//     PlcTask Inputs/GVL_iXlinker.EtherCAT_Master_EPPxxxx.Beckhoff_EPP2xxx.Beckhoff_EPP2xxxEK1122.A_0083_EPP2817_0008_0018.DIG_Diag_Inputs_Channel_2.Diag_Input[1] <-> DIG Diag Inputs Channel 2/Diag Input 2
//     PlcTask Inputs/GVL_iXlinker.EtherCAT_Master_EPPxxxx.Beckhoff_EPP2xxx.Beckhoff_EPP2xxxEK1122.A_0083_EPP2817_0008_0018.DIG_Diag_Inputs_Channel_2.Diag_Input[2] <-> DIG Diag Inputs Channel 2/Diag Input 3
//     PlcTask Inputs/GVL_iXlinker.EtherCAT_Master_EPPxxxx.Beckhoff_EPP2xxx.Beckhoff_EPP2xxxEK1122.A_0083_EPP2817_0008_0018.DIG_Diag_Inputs_Channel_2.Diag_Input[3] <-> DIG Diag Inputs Channel 2/Diag Input 4
//     PlcTask Inputs/GVL_iXlinker.EtherCAT_Master_EPPxxxx.Beckhoff_EPP2xxx.Beckhoff_EPP2xxxEK1122.A_0083_EPP2817_0008_0018.DIG_Diag_Inputs_Channel_2.Diag_Input[4] <-> DIG Diag Inputs Channel 2/Diag Input 5
//     PlcTask Inputs/GVL_iXlinker.EtherCAT_Master_EPPxxxx.Beckhoff_EPP2xxx.Beckhoff_EPP2xxxEK1122.A_0083_EPP2817_0008_0018.DIG_Diag_Inputs_Channel_2.Diag_Input[5] <-> DIG Diag Inputs Channel 2/Diag Input 6
//     PlcTask Inputs/GVL_iXlinker.EtherCAT_Master_EPPxxxx.Beckhoff_EPP2xxx.Beckhoff_EPP2xxxEK1122.A_0083_EPP2817_0008_0018.DIG_Diag_Inputs_Channel_2.Diag_Input[6] <-> DIG Diag Inputs Channel 2/Diag Input 7
//     PlcTask Inputs/GVL_iXlinker.EtherCAT_Master_EPPxxxx.Beckhoff_EPP2xxx.Beckhoff_EPP2xxxEK1122.A_0083_EPP2817_0008_0018.DIG_Diag_Inputs_Channel_2.Diag_Input[7] <-> DIG Diag Inputs Channel 2/Diag Input 8
//     PlcTask Inputs/GVL_iXlinker.EtherCAT_Master_EPPxxxx.Beckhoff_EPP2xxx.Beckhoff_EPP2xxxEK1122.A_0083_EPP2817_0008_0018.DIG_Diag_Inputs_Channel_3.Diag_Input[0] <-> DIG Diag Inputs Channel 3/Diag Input 1
//     PlcTask Inputs/GVL_iXlinker.EtherCAT_Master_EPPxxxx.Beckhoff_EPP2xxx.Beckhoff_EPP2xxxEK1122.A_0083_EPP2817_0008_0018.DIG_Diag_Inputs_Channel_3.Diag_Input[1] <-> DIG Diag Inputs Channel 3/Diag Input 2
//     PlcTask Inputs/GVL_iXlinker.EtherCAT_Master_EPPxxxx.Beckhoff_EPP2xxx.Beckhoff_EPP2xxxEK1122.A_0083_EPP2817_0008_0018.DIG_Diag_Inputs_Channel_3.Diag_Input[2] <-> DIG Diag Inputs Channel 3/Diag Input 3
//     PlcTask Inputs/GVL_iXlinker.EtherCAT_Master_EPPxxxx.Beckhoff_EPP2xxx.Beckhoff_EPP2xxxEK1122.A_0083_EPP2817_0008_0018.DIG_Diag_Inputs_Channel_3.Diag_Input[3] <-> DIG Diag Inputs Channel 3/Diag Input 4
//     PlcTask Inputs/GVL_iXlinker.EtherCAT_Master_EPPxxxx.Beckhoff_EPP2xxx.Beckhoff_EPP2xxxEK1122.A_0083_EPP2817_0008_0018.DIG_Diag_Inputs_Channel_3.Diag_Input[4] <-> DIG Diag Inputs Channel 3/Diag Input 5
//     PlcTask Inputs/GVL_iXlinker.EtherCAT_Master_EPPxxxx.Beckhoff_EPP2xxx.Beckhoff_EPP2xxxEK1122.A_0083_EPP2817_0008_0018.DIG_Diag_Inputs_Channel_3.Diag_Input[5] <-> DIG Diag Inputs Channel 3/Diag Input 6
//     PlcTask Inputs/GVL_iXlinker.EtherCAT_Master_EPPxxxx.Beckhoff_EPP2xxx.Beckhoff_EPP2xxxEK1122.A_0083_EPP2817_0008_0018.DIG_Diag_Inputs_Channel_3.Diag_Input[6] <-> DIG Diag Inputs Channel 3/Diag Input 7
//     PlcTask Inputs/GVL_iXlinker.EtherCAT_Master_EPPxxxx.Beckhoff_EPP2xxx.Beckhoff_EPP2xxxEK1122.A_0083_EPP2817_0008_0018.DIG_Diag_Inputs_Channel_3.Diag_Input[7] <-> DIG Diag Inputs Channel 3/Diag Input 8
//     PlcTask Inputs/GVL_iXlinker.EtherCAT_Master_EPPxxxx.Beckhoff_EPP2xxx.Beckhoff_EPP2xxxEK1122.A_0083_EPP2817_0008_0018.DIG_Inputs_Device.Safe_state_active <-> DIG Inputs Device/Safe state active
//     PlcTask Inputs/GVL_iXlinker.EtherCAT_Master_EPPxxxx.Beckhoff_EPP2xxx.Beckhoff_EPP2xxxEK1122.A_0083_EPP2817_0008_0018.DIG_Inputs_Device.Error_channel[0] <-> DIG Inputs Device/Error channel 1
//     PlcTask Inputs/GVL_iXlinker.EtherCAT_Master_EPPxxxx.Beckhoff_EPP2xxx.Beckhoff_EPP2xxxEK1122.A_0083_EPP2817_0008_0018.DIG_Inputs_Device.Error_channel[1] <-> DIG Inputs Device/Error channel 2
//     PlcTask Inputs/GVL_iXlinker.EtherCAT_Master_EPPxxxx.Beckhoff_EPP2xxx.Beckhoff_EPP2xxxEK1122.A_0083_EPP2817_0008_0018.DIG_Inputs_Device.Error_channel[2] <-> DIG Inputs Device/Error channel 3
//     PlcTask Inputs/GVL_iXlinker.EtherCAT_Master_EPPxxxx.Beckhoff_EPP2xxx.Beckhoff_EPP2xxxEK1122.A_0083_EPP2817_0008_0018.DIG_Inputs_Device.Us_Undervoltage <-> DIG Inputs Device/Us Undervoltage
//     PlcTask Inputs/GVL_iXlinker.EtherCAT_Master_EPPxxxx.Beckhoff_EPP2xxx.Beckhoff_EPP2xxxEK1122.A_0083_EPP2817_0008_0018.DIG_Inputs_Device.Up_Undervoltage <-> DIG Inputs Device/Up Undervoltage
//     PlcTask Inputs/GVL_iXlinker.EtherCAT_Master_EPPxxxx.Beckhoff_EPP2xxx.Beckhoff_EPP2xxxEK1122.A_0083_EPP2817_0008_0018.DIG_Inputs_Device.Sync_error <-> DIG Inputs Device/Sync error
//     PlcTask Inputs/GVL_iXlinker.EtherCAT_Master_EPPxxxx.Beckhoff_EPP2xxx.Beckhoff_EPP2xxxEK1122.A_0083_EPP2817_0008_0018.DIG_Inputs_Device.TxPDO_Toggle <-> DIG Inputs Device/TxPDO Toggle
//     PlcTask Outputs/GVL_iXlinker.EtherCAT_Master_EPPxxxx.Beckhoff_EPP2xxx.Beckhoff_EPP2xxxEK1122.A_0083_EPP2817_0008_0018.DIG_Output_Channel_1.Output[0] <-> DIG Output Channel 1/Output 1
//     PlcTask Outputs/GVL_iXlinker.EtherCAT_Master_EPPxxxx.Beckhoff_EPP2xxx.Beckhoff_EPP2xxxEK1122.A_0083_EPP2817_0008_0018.DIG_Output_Channel_1.Output[1] <-> DIG Output Channel 1/Output 2
//     PlcTask Outputs/GVL_iXlinker.EtherCAT_Master_EPPxxxx.Beckhoff_EPP2xxx.Beckhoff_EPP2xxxEK1122.A_0083_EPP2817_0008_0018.DIG_Output_Channel_1.Output[2] <-> DIG Output Channel 1/Output 3
//     PlcTask Outputs/GVL_iXlinker.EtherCAT_Master_EPPxxxx.Beckhoff_EPP2xxx.Beckhoff_EPP2xxxEK1122.A_0083_EPP2817_0008_0018.DIG_Output_Channel_1.Output[3] <-> DIG Output Channel 1/Output 4
//     PlcTask Outputs/GVL_iXlinker.EtherCAT_Master_EPPxxxx.Beckhoff_EPP2xxx.Beckhoff_EPP2xxxEK1122.A_0083_EPP2817_0008_0018.DIG_Output_Channel_1.Output[4] <-> DIG Output Channel 1/Output 5
//     PlcTask Outputs/GVL_iXlinker.EtherCAT_Master_EPPxxxx.Beckhoff_EPP2xxx.Beckhoff_EPP2xxxEK1122.A_0083_EPP2817_0008_0018.DIG_Output_Channel_1.Output[5] <-> DIG Output Channel 1/Output 6
//     PlcTask Outputs/GVL_iXlinker.EtherCAT_Master_EPPxxxx.Beckhoff_EPP2xxx.Beckhoff_EPP2xxxEK1122.A_0083_EPP2817_0008_0018.DIG_Output_Channel_1.Output[6] <-> DIG Output Channel 1/Output 7
//     PlcTask Outputs/GVL_iXlinker.EtherCAT_Master_EPPxxxx.Beckhoff_EPP2xxx.Beckhoff_EPP2xxxEK1122.A_0083_EPP2817_0008_0018.DIG_Output_Channel_1.Output[7] <-> DIG Output Channel 1/Output 8
//     PlcTask Outputs/GVL_iXlinker.EtherCAT_Master_EPPxxxx.Beckhoff_EPP2xxx.Beckhoff_EPP2xxxEK1122.A_0083_EPP2817_0008_0018.DIG_Output_Channel_2.Output[0] <-> DIG Output Channel 2/Output 1
//     PlcTask Outputs/GVL_iXlinker.EtherCAT_Master_EPPxxxx.Beckhoff_EPP2xxx.Beckhoff_EPP2xxxEK1122.A_0083_EPP2817_0008_0018.DIG_Output_Channel_2.Output[1] <-> DIG Output Channel 2/Output 2
//     PlcTask Outputs/GVL_iXlinker.EtherCAT_Master_EPPxxxx.Beckhoff_EPP2xxx.Beckhoff_EPP2xxxEK1122.A_0083_EPP2817_0008_0018.DIG_Output_Channel_2.Output[2] <-> DIG Output Channel 2/Output 3
//     PlcTask Outputs/GVL_iXlinker.EtherCAT_Master_EPPxxxx.Beckhoff_EPP2xxx.Beckhoff_EPP2xxxEK1122.A_0083_EPP2817_0008_0018.DIG_Output_Channel_2.Output[3] <-> DIG Output Channel 2/Output 4
//     PlcTask Outputs/GVL_iXlinker.EtherCAT_Master_EPPxxxx.Beckhoff_EPP2xxx.Beckhoff_EPP2xxxEK1122.A_0083_EPP2817_0008_0018.DIG_Output_Channel_2.Output[4] <-> DIG Output Channel 2/Output 5
//     PlcTask Outputs/GVL_iXlinker.EtherCAT_Master_EPPxxxx.Beckhoff_EPP2xxx.Beckhoff_EPP2xxxEK1122.A_0083_EPP2817_0008_0018.DIG_Output_Channel_2.Output[5] <-> DIG Output Channel 2/Output 6
//     PlcTask Outputs/GVL_iXlinker.EtherCAT_Master_EPPxxxx.Beckhoff_EPP2xxx.Beckhoff_EPP2xxxEK1122.A_0083_EPP2817_0008_0018.DIG_Output_Channel_2.Output[6] <-> DIG Output Channel 2/Output 7
//     PlcTask Outputs/GVL_iXlinker.EtherCAT_Master_EPPxxxx.Beckhoff_EPP2xxx.Beckhoff_EPP2xxxEK1122.A_0083_EPP2817_0008_0018.DIG_Output_Channel_2.Output[7] <-> DIG Output Channel 2/Output 8
//     PlcTask Outputs/GVL_iXlinker.EtherCAT_Master_EPPxxxx.Beckhoff_EPP2xxx.Beckhoff_EPP2xxxEK1122.A_0083_EPP2817_0008_0018.DIG_Output_Channel_3.Output[0] <-> DIG Output Channel 3/Output 1
//     PlcTask Outputs/GVL_iXlinker.EtherCAT_Master_EPPxxxx.Beckhoff_EPP2xxx.Beckhoff_EPP2xxxEK1122.A_0083_EPP2817_0008_0018.DIG_Output_Channel_3.Output[1] <-> DIG Output Channel 3/Output 2
//     PlcTask Outputs/GVL_iXlinker.EtherCAT_Master_EPPxxxx.Beckhoff_EPP2xxx.Beckhoff_EPP2xxxEK1122.A_0083_EPP2817_0008_0018.DIG_Output_Channel_3.Output[2] <-> DIG Output Channel 3/Output 3
//     PlcTask Outputs/GVL_iXlinker.EtherCAT_Master_EPPxxxx.Beckhoff_EPP2xxx.Beckhoff_EPP2xxxEK1122.A_0083_EPP2817_0008_0018.DIG_Output_Channel_3.Output[3] <-> DIG Output Channel 3/Output 4
//     PlcTask Outputs/GVL_iXlinker.EtherCAT_Master_EPPxxxx.Beckhoff_EPP2xxx.Beckhoff_EPP2xxxEK1122.A_0083_EPP2817_0008_0018.DIG_Output_Channel_3.Output[4] <-> DIG Output Channel 3/Output 5
//     PlcTask Outputs/GVL_iXlinker.EtherCAT_Master_EPPxxxx.Beckhoff_EPP2xxx.Beckhoff_EPP2xxxEK1122.A_0083_EPP2817_0008_0018.DIG_Output_Channel_3.Output[5] <-> DIG Output Channel 3/Output 6
//     PlcTask Outputs/GVL_iXlinker.EtherCAT_Master_EPPxxxx.Beckhoff_EPP2xxx.Beckhoff_EPP2xxxEK1122.A_0083_EPP2817_0008_0018.DIG_Output_Channel_3.Output[6] <-> DIG Output Channel 3/Output 7
//     PlcTask Outputs/GVL_iXlinker.EtherCAT_Master_EPPxxxx.Beckhoff_EPP2xxx.Beckhoff_EPP2xxxEK1122.A_0083_EPP2817_0008_0018.DIG_Output_Channel_3.Output[7] <-> DIG Output Channel 3/Output 8
//     PlcTask Outputs/GVL_iXlinker.EtherCAT_Master_EPPxxxx.Beckhoff_EPP2xxx.Beckhoff_EPP2xxxEK1122.A_0083_EPP2817_0008_0018.DIG_Outputs_Device.Set_safe_state <-> DIG Outputs Device/Set safe state
//     PlcTask Outputs/GVL_iXlinker.EtherCAT_Master_EPPxxxx.Beckhoff_EPP2xxx.Beckhoff_EPP2xxxEK1122.A_0083_EPP2817_0008_0018.DIG_Outputs_Device.Reset_outputs <-> DIG Outputs Device/Reset outputs
//     PlcTask Inputs/GVL_iXlinker.EtherCAT_Master_EPPxxxx.Beckhoff_EPP2xxx.Beckhoff_EPP2xxxEK1122.A_0083_EPP2817_0008_0018.WcState.WcState <-> WcState/WcState
//     PlcTask Inputs/GVL_iXlinker.EtherCAT_Master_EPPxxxx.Beckhoff_EPP2xxx.Beckhoff_EPP2xxxEK1122.A_0083_EPP2817_0008_0018.WcState.InputToggle <-> WcState/InputToggle
//     PlcTask Inputs/GVL_iXlinker.EtherCAT_Master_EPPxxxx.Beckhoff_EPP2xxx.Beckhoff_EPP2xxxEK1122.A_0083_EPP2817_0008_0018.InfoData.AdsAddr <-> InfoData/AdsAddr
//     PlcTask Inputs/GVL_iXlinker.EtherCAT_Master_EPPxxxx.Beckhoff_EPP2xxx.Beckhoff_EPP2xxxEK1122.A_0083_EPP2817_0008_0018.InfoData.State <-> InfoData/State
//   PLC/PLC Instance <-> EtherCAT Master EPPxxxx/Beckhoff EPP3xxx
//     PlcTask Inputs/GVL_iXlinker.EtherCAT_Master_EPPxxxx.Beckhoff_EPP3xxx.InfoData.State <-> InfoData/State
//   PLC/PLC Instance <-> EtherCAT Master EPPxxxx/Beckhoff EPP3xxx/Beckhoff EPP3xxxEK1122
//     PlcTask Inputs/GVL_iXlinker.EtherCAT_Master_EPPxxxx.Beckhoff_EPP3xxx.Beckhoff_EPP3xxxEK1122.InfoData.State <-> InfoData/State
//   PLC/PLC Instance <-> EtherCAT Master EPPxxxx/Beckhoff EPP3xxx/Beckhoff EPP3xxxEK1122/Beckhoff EPP3xxxsub EK1100
//     PlcTask Inputs/GVL_iXlinker.EtherCAT_Master_EPPxxxx.Beckhoff_EPP3xxx.Beckhoff_EPP3xxxEK1122.Beckhoff_EPP3xxxsub_EK1100.InfoData.State <-> InfoData/State
//   PLC/PLC Instance <-> EtherCAT Master EPPxxxx/Beckhoff EPP3xxx/Beckhoff EPP3xxxEK1122/A_0001(EPP3174-0002-0016)
//     PlcTask Inputs/GVL_iXlinker.EtherCAT_Master_EPPxxxx.Beckhoff_EPP3xxx.Beckhoff_EPP3xxxEK1122.A_0001_EPP3174_0002_0016.AI_Standard_Channel_1.Status/Underrange <-> AI Standard Channel 1/Status/Underrange
//     PlcTask Inputs/GVL_iXlinker.EtherCAT_Master_EPPxxxx.Beckhoff_EPP3xxx.Beckhoff_EPP3xxxEK1122.A_0001_EPP3174_0002_0016.AI_Standard_Channel_2.Status/Underrange <-> AI Standard Channel 2/Status/Underrange
//     PlcTask Inputs/GVL_iXlinker.EtherCAT_Master_EPPxxxx.Beckhoff_EPP3xxx.Beckhoff_EPP3xxxEK1122.A_0001_EPP3174_0002_0016.AI_Standard_Channel_3.Status/Underrange <-> AI Standard Channel 3/Status/Underrange
//     PlcTask Inputs/GVL_iXlinker.EtherCAT_Master_EPPxxxx.Beckhoff_EPP3xxx.Beckhoff_EPP3xxxEK1122.A_0001_EPP3174_0002_0016.AI_Standard_Channel_4.Status/Underrange <-> AI Standard Channel 4/Status/Underrange
//     PlcTask Inputs/GVL_iXlinker.EtherCAT_Master_EPPxxxx.Beckhoff_EPP3xxx.Beckhoff_EPP3xxxEK1122.A_0001_EPP3174_0002_0016.AI_Standard_Channel_1.Status/Overrange <-> AI Standard Channel 1/Status/Overrange
//     PlcTask Inputs/GVL_iXlinker.EtherCAT_Master_EPPxxxx.Beckhoff_EPP3xxx.Beckhoff_EPP3xxxEK1122.A_0001_EPP3174_0002_0016.AI_Standard_Channel_2.Status/Overrange <-> AI Standard Channel 2/Status/Overrange
//     PlcTask Inputs/GVL_iXlinker.EtherCAT_Master_EPPxxxx.Beckhoff_EPP3xxx.Beckhoff_EPP3xxxEK1122.A_0001_EPP3174_0002_0016.AI_Standard_Channel_3.Status/Overrange <-> AI Standard Channel 3/Status/Overrange
//     PlcTask Inputs/GVL_iXlinker.EtherCAT_Master_EPPxxxx.Beckhoff_EPP3xxx.Beckhoff_EPP3xxxEK1122.A_0001_EPP3174_0002_0016.AI_Standard_Channel_4.Status/Overrange <-> AI Standard Channel 4/Status/Overrange
//     PlcTask Inputs/GVL_iXlinker.EtherCAT_Master_EPPxxxx.Beckhoff_EPP3xxx.Beckhoff_EPP3xxxEK1122.A_0001_EPP3174_0002_0016.AI_Standard_Channel_1.Status/Limit_1 <-> AI Standard Channel 1/Status/Limit 1
//     PlcTask Inputs/GVL_iXlinker.EtherCAT_Master_EPPxxxx.Beckhoff_EPP3xxx.Beckhoff_EPP3xxxEK1122.A_0001_EPP3174_0002_0016.AI_Standard_Channel_1.Status/Limit_2 <-> AI Standard Channel 1/Status/Limit 2
//     PlcTask Inputs/GVL_iXlinker.EtherCAT_Master_EPPxxxx.Beckhoff_EPP3xxx.Beckhoff_EPP3xxxEK1122.A_0001_EPP3174_0002_0016.AI_Standard_Channel_2.Status/Limit_1 <-> AI Standard Channel 2/Status/Limit 1
//     PlcTask Inputs/GVL_iXlinker.EtherCAT_Master_EPPxxxx.Beckhoff_EPP3xxx.Beckhoff_EPP3xxxEK1122.A_0001_EPP3174_0002_0016.AI_Standard_Channel_2.Status/Limit_2 <-> AI Standard Channel 2/Status/Limit 2
//     PlcTask Inputs/GVL_iXlinker.EtherCAT_Master_EPPxxxx.Beckhoff_EPP3xxx.Beckhoff_EPP3xxxEK1122.A_0001_EPP3174_0002_0016.AI_Standard_Channel_3.Status/Limit_1 <-> AI Standard Channel 3/Status/Limit 1
//     PlcTask Inputs/GVL_iXlinker.EtherCAT_Master_EPPxxxx.Beckhoff_EPP3xxx.Beckhoff_EPP3xxxEK1122.A_0001_EPP3174_0002_0016.AI_Standard_Channel_3.Status/Limit_2 <-> AI Standard Channel 3/Status/Limit 2
//     PlcTask Inputs/GVL_iXlinker.EtherCAT_Master_EPPxxxx.Beckhoff_EPP3xxx.Beckhoff_EPP3xxxEK1122.A_0001_EPP3174_0002_0016.AI_Standard_Channel_4.Status/Limit_1 <-> AI Standard Channel 4/Status/Limit 1
//     PlcTask Inputs/GVL_iXlinker.EtherCAT_Master_EPPxxxx.Beckhoff_EPP3xxx.Beckhoff_EPP3xxxEK1122.A_0001_EPP3174_0002_0016.AI_Standard_Channel_4.Status/Limit_2 <-> AI Standard Channel 4/Status/Limit 2
//     PlcTask Inputs/GVL_iXlinker.EtherCAT_Master_EPPxxxx.Beckhoff_EPP3xxx.Beckhoff_EPP3xxxEK1122.A_0001_EPP3174_0002_0016.AI_Standard_Channel_1.Status/Error <-> AI Standard Channel 1/Status/Error
//     PlcTask Inputs/GVL_iXlinker.EtherCAT_Master_EPPxxxx.Beckhoff_EPP3xxx.Beckhoff_EPP3xxxEK1122.A_0001_EPP3174_0002_0016.AI_Standard_Channel_2.Status/Error <-> AI Standard Channel 2/Status/Error
//     PlcTask Inputs/GVL_iXlinker.EtherCAT_Master_EPPxxxx.Beckhoff_EPP3xxx.Beckhoff_EPP3xxxEK1122.A_0001_EPP3174_0002_0016.AI_Standard_Channel_3.Status/Error <-> AI Standard Channel 3/Status/Error
//     PlcTask Inputs/GVL_iXlinker.EtherCAT_Master_EPPxxxx.Beckhoff_EPP3xxx.Beckhoff_EPP3xxxEK1122.A_0001_EPP3174_0002_0016.AI_Standard_Channel_4.Status/Error <-> AI Standard Channel 4/Status/Error
//     PlcTask Inputs/GVL_iXlinker.EtherCAT_Master_EPPxxxx.Beckhoff_EPP3xxx.Beckhoff_EPP3xxxEK1122.A_0001_EPP3174_0002_0016.AI_Standard_Channel_1.Status/Sync_error <-> AI Standard Channel 1/Status/Sync error
//     PlcTask Inputs/GVL_iXlinker.EtherCAT_Master_EPPxxxx.Beckhoff_EPP3xxx.Beckhoff_EPP3xxxEK1122.A_0001_EPP3174_0002_0016.AI_Standard_Channel_2.Status/Sync_error <-> AI Standard Channel 2/Status/Sync error
//     PlcTask Inputs/GVL_iXlinker.EtherCAT_Master_EPPxxxx.Beckhoff_EPP3xxx.Beckhoff_EPP3xxxEK1122.A_0001_EPP3174_0002_0016.AI_Standard_Channel_3.Status/Sync_error <-> AI Standard Channel 3/Status/Sync error
//     PlcTask Inputs/GVL_iXlinker.EtherCAT_Master_EPPxxxx.Beckhoff_EPP3xxx.Beckhoff_EPP3xxxEK1122.A_0001_EPP3174_0002_0016.AI_Standard_Channel_4.Status/Sync_error <-> AI Standard Channel 4/Status/Sync error
//     PlcTask Inputs/GVL_iXlinker.EtherCAT_Master_EPPxxxx.Beckhoff_EPP3xxx.Beckhoff_EPP3xxxEK1122.A_0001_EPP3174_0002_0016.AI_Standard_Channel_1.Status/TxPDO_State <-> AI Standard Channel 1/Status/TxPDO State
//     PlcTask Inputs/GVL_iXlinker.EtherCAT_Master_EPPxxxx.Beckhoff_EPP3xxx.Beckhoff_EPP3xxxEK1122.A_0001_EPP3174_0002_0016.AI_Standard_Channel_2.Status/TxPDO_State <-> AI Standard Channel 2/Status/TxPDO State
//     PlcTask Inputs/GVL_iXlinker.EtherCAT_Master_EPPxxxx.Beckhoff_EPP3xxx.Beckhoff_EPP3xxxEK1122.A_0001_EPP3174_0002_0016.AI_Standard_Channel_3.Status/TxPDO_State <-> AI Standard Channel 3/Status/TxPDO State
//     PlcTask Inputs/GVL_iXlinker.EtherCAT_Master_EPPxxxx.Beckhoff_EPP3xxx.Beckhoff_EPP3xxxEK1122.A_0001_EPP3174_0002_0016.AI_Standard_Channel_4.Status/TxPDO_State <-> AI Standard Channel 4/Status/TxPDO State
//     PlcTask Inputs/GVL_iXlinker.EtherCAT_Master_EPPxxxx.Beckhoff_EPP3xxx.Beckhoff_EPP3xxxEK1122.A_0001_EPP3174_0002_0016.AI_Standard_Channel_1.Status/TxPDO_Toggle <-> AI Standard Channel 1/Status/TxPDO Toggle
//     PlcTask Inputs/GVL_iXlinker.EtherCAT_Master_EPPxxxx.Beckhoff_EPP3xxx.Beckhoff_EPP3xxxEK1122.A_0001_EPP3174_0002_0016.AI_Standard_Channel_2.Status/TxPDO_Toggle <-> AI Standard Channel 2/Status/TxPDO Toggle
//     PlcTask Inputs/GVL_iXlinker.EtherCAT_Master_EPPxxxx.Beckhoff_EPP3xxx.Beckhoff_EPP3xxxEK1122.A_0001_EPP3174_0002_0016.AI_Standard_Channel_3.Status/TxPDO_Toggle <-> AI Standard Channel 3/Status/TxPDO Toggle
//     PlcTask Inputs/GVL_iXlinker.EtherCAT_Master_EPPxxxx.Beckhoff_EPP3xxx.Beckhoff_EPP3xxxEK1122.A_0001_EPP3174_0002_0016.AI_Standard_Channel_4.Status/TxPDO_Toggle <-> AI Standard Channel 4/Status/TxPDO Toggle
//     PlcTask Inputs/GVL_iXlinker.EtherCAT_Master_EPPxxxx.Beckhoff_EPP3xxx.Beckhoff_EPP3xxxEK1122.A_0001_EPP3174_0002_0016.AI_Standard_Channel_1.Value <-> AI Standard Channel 1/Value
//     PlcTask Inputs/GVL_iXlinker.EtherCAT_Master_EPPxxxx.Beckhoff_EPP3xxx.Beckhoff_EPP3xxxEK1122.A_0001_EPP3174_0002_0016.AI_Standard_Channel_2.Value <-> AI Standard Channel 2/Value
//     PlcTask Inputs/GVL_iXlinker.EtherCAT_Master_EPPxxxx.Beckhoff_EPP3xxx.Beckhoff_EPP3xxxEK1122.A_0001_EPP3174_0002_0016.AI_Standard_Channel_3.Value <-> AI Standard Channel 3/Value
//     PlcTask Inputs/GVL_iXlinker.EtherCAT_Master_EPPxxxx.Beckhoff_EPP3xxx.Beckhoff_EPP3xxxEK1122.A_0001_EPP3174_0002_0016.AI_Standard_Channel_4.Value <-> AI Standard Channel 4/Value
//     PlcTask Inputs/GVL_iXlinker.EtherCAT_Master_EPPxxxx.Beckhoff_EPP3xxx.Beckhoff_EPP3xxxEK1122.A_0001_EPP3174_0002_0016.WcState.WcState <-> WcState/WcState
//     PlcTask Inputs/GVL_iXlinker.EtherCAT_Master_EPPxxxx.Beckhoff_EPP3xxx.Beckhoff_EPP3xxxEK1122.A_0001_EPP3174_0002_0016.WcState.InputToggle <-> WcState/InputToggle
//     PlcTask Inputs/GVL_iXlinker.EtherCAT_Master_EPPxxxx.Beckhoff_EPP3xxx.Beckhoff_EPP3xxxEK1122.A_0001_EPP3174_0002_0016.InfoData.AdsAddr <-> InfoData/AdsAddr
//     PlcTask Inputs/GVL_iXlinker.EtherCAT_Master_EPPxxxx.Beckhoff_EPP3xxx.Beckhoff_EPP3xxxEK1122.A_0001_EPP3174_0002_0016.InfoData.State <-> InfoData/State
//   PLC/PLC Instance <-> EtherCAT Master EPPxxxx/Beckhoff EPP3xxx/Beckhoff EPP3xxxEK1122/A_0002(EPP3174-0002-0017)
//     PlcTask Inputs/GVL_iXlinker.EtherCAT_Master_EPPxxxx.Beckhoff_EPP3xxx.Beckhoff_EPP3xxxEK1122.A_0002_EPP3174_0002_0017.AI_Standard_Channel_1.Status/Underrange <-> AI Standard Channel 1/Status/Underrange
//     PlcTask Inputs/GVL_iXlinker.EtherCAT_Master_EPPxxxx.Beckhoff_EPP3xxx.Beckhoff_EPP3xxxEK1122.A_0002_EPP3174_0002_0017.AI_Standard_Channel_2.Status/Underrange <-> AI Standard Channel 2/Status/Underrange
//     PlcTask Inputs/GVL_iXlinker.EtherCAT_Master_EPPxxxx.Beckhoff_EPP3xxx.Beckhoff_EPP3xxxEK1122.A_0002_EPP3174_0002_0017.AI_Standard_Channel_3.Status/Underrange <-> AI Standard Channel 3/Status/Underrange
//     PlcTask Inputs/GVL_iXlinker.EtherCAT_Master_EPPxxxx.Beckhoff_EPP3xxx.Beckhoff_EPP3xxxEK1122.A_0002_EPP3174_0002_0017.AI_Standard_Channel_4.Status/Underrange <-> AI Standard Channel 4/Status/Underrange
//     PlcTask Inputs/GVL_iXlinker.EtherCAT_Master_EPPxxxx.Beckhoff_EPP3xxx.Beckhoff_EPP3xxxEK1122.A_0002_EPP3174_0002_0017.AI_Standard_Channel_1.Status/Overrange <-> AI Standard Channel 1/Status/Overrange
//     PlcTask Inputs/GVL_iXlinker.EtherCAT_Master_EPPxxxx.Beckhoff_EPP3xxx.Beckhoff_EPP3xxxEK1122.A_0002_EPP3174_0002_0017.AI_Standard_Channel_2.Status/Overrange <-> AI Standard Channel 2/Status/Overrange
//     PlcTask Inputs/GVL_iXlinker.EtherCAT_Master_EPPxxxx.Beckhoff_EPP3xxx.Beckhoff_EPP3xxxEK1122.A_0002_EPP3174_0002_0017.AI_Standard_Channel_3.Status/Overrange <-> AI Standard Channel 3/Status/Overrange
//     PlcTask Inputs/GVL_iXlinker.EtherCAT_Master_EPPxxxx.Beckhoff_EPP3xxx.Beckhoff_EPP3xxxEK1122.A_0002_EPP3174_0002_0017.AI_Standard_Channel_4.Status/Overrange <-> AI Standard Channel 4/Status/Overrange
//     PlcTask Inputs/GVL_iXlinker.EtherCAT_Master_EPPxxxx.Beckhoff_EPP3xxx.Beckhoff_EPP3xxxEK1122.A_0002_EPP3174_0002_0017.AI_Standard_Channel_1.Status/Limit_1 <-> AI Standard Channel 1/Status/Limit 1
//     PlcTask Inputs/GVL_iXlinker.EtherCAT_Master_EPPxxxx.Beckhoff_EPP3xxx.Beckhoff_EPP3xxxEK1122.A_0002_EPP3174_0002_0017.AI_Standard_Channel_1.Status/Limit_2 <-> AI Standard Channel 1/Status/Limit 2
//     PlcTask Inputs/GVL_iXlinker.EtherCAT_Master_EPPxxxx.Beckhoff_EPP3xxx.Beckhoff_EPP3xxxEK1122.A_0002_EPP3174_0002_0017.AI_Standard_Channel_2.Status/Limit_1 <-> AI Standard Channel 2/Status/Limit 1
//     PlcTask Inputs/GVL_iXlinker.EtherCAT_Master_EPPxxxx.Beckhoff_EPP3xxx.Beckhoff_EPP3xxxEK1122.A_0002_EPP3174_0002_0017.AI_Standard_Channel_2.Status/Limit_2 <-> AI Standard Channel 2/Status/Limit 2
//     PlcTask Inputs/GVL_iXlinker.EtherCAT_Master_EPPxxxx.Beckhoff_EPP3xxx.Beckhoff_EPP3xxxEK1122.A_0002_EPP3174_0002_0017.AI_Standard_Channel_3.Status/Limit_1 <-> AI Standard Channel 3/Status/Limit 1
//     PlcTask Inputs/GVL_iXlinker.EtherCAT_Master_EPPxxxx.Beckhoff_EPP3xxx.Beckhoff_EPP3xxxEK1122.A_0002_EPP3174_0002_0017.AI_Standard_Channel_3.Status/Limit_2 <-> AI Standard Channel 3/Status/Limit 2
//     PlcTask Inputs/GVL_iXlinker.EtherCAT_Master_EPPxxxx.Beckhoff_EPP3xxx.Beckhoff_EPP3xxxEK1122.A_0002_EPP3174_0002_0017.AI_Standard_Channel_4.Status/Limit_1 <-> AI Standard Channel 4/Status/Limit 1
//     PlcTask Inputs/GVL_iXlinker.EtherCAT_Master_EPPxxxx.Beckhoff_EPP3xxx.Beckhoff_EPP3xxxEK1122.A_0002_EPP3174_0002_0017.AI_Standard_Channel_4.Status/Limit_2 <-> AI Standard Channel 4/Status/Limit 2
//     PlcTask Inputs/GVL_iXlinker.EtherCAT_Master_EPPxxxx.Beckhoff_EPP3xxx.Beckhoff_EPP3xxxEK1122.A_0002_EPP3174_0002_0017.AI_Standard_Channel_1.Status/Error <-> AI Standard Channel 1/Status/Error
//     PlcTask Inputs/GVL_iXlinker.EtherCAT_Master_EPPxxxx.Beckhoff_EPP3xxx.Beckhoff_EPP3xxxEK1122.A_0002_EPP3174_0002_0017.AI_Standard_Channel_2.Status/Error <-> AI Standard Channel 2/Status/Error
//     PlcTask Inputs/GVL_iXlinker.EtherCAT_Master_EPPxxxx.Beckhoff_EPP3xxx.Beckhoff_EPP3xxxEK1122.A_0002_EPP3174_0002_0017.AI_Standard_Channel_3.Status/Error <-> AI Standard Channel 3/Status/Error
//     PlcTask Inputs/GVL_iXlinker.EtherCAT_Master_EPPxxxx.Beckhoff_EPP3xxx.Beckhoff_EPP3xxxEK1122.A_0002_EPP3174_0002_0017.AI_Standard_Channel_4.Status/Error <-> AI Standard Channel 4/Status/Error
//     PlcTask Inputs/GVL_iXlinker.EtherCAT_Master_EPPxxxx.Beckhoff_EPP3xxx.Beckhoff_EPP3xxxEK1122.A_0002_EPP3174_0002_0017.AI_Standard_Channel_1.Status/Sync_error <-> AI Standard Channel 1/Status/Sync error
//     PlcTask Inputs/GVL_iXlinker.EtherCAT_Master_EPPxxxx.Beckhoff_EPP3xxx.Beckhoff_EPP3xxxEK1122.A_0002_EPP3174_0002_0017.AI_Standard_Channel_2.Status/Sync_error <-> AI Standard Channel 2/Status/Sync error
//     PlcTask Inputs/GVL_iXlinker.EtherCAT_Master_EPPxxxx.Beckhoff_EPP3xxx.Beckhoff_EPP3xxxEK1122.A_0002_EPP3174_0002_0017.AI_Standard_Channel_3.Status/Sync_error <-> AI Standard Channel 3/Status/Sync error
//     PlcTask Inputs/GVL_iXlinker.EtherCAT_Master_EPPxxxx.Beckhoff_EPP3xxx.Beckhoff_EPP3xxxEK1122.A_0002_EPP3174_0002_0017.AI_Standard_Channel_4.Status/Sync_error <-> AI Standard Channel 4/Status/Sync error
//     PlcTask Inputs/GVL_iXlinker.EtherCAT_Master_EPPxxxx.Beckhoff_EPP3xxx.Beckhoff_EPP3xxxEK1122.A_0002_EPP3174_0002_0017.AI_Standard_Channel_1.Status/TxPDO_State <-> AI Standard Channel 1/Status/TxPDO State
//     PlcTask Inputs/GVL_iXlinker.EtherCAT_Master_EPPxxxx.Beckhoff_EPP3xxx.Beckhoff_EPP3xxxEK1122.A_0002_EPP3174_0002_0017.AI_Standard_Channel_2.Status/TxPDO_State <-> AI Standard Channel 2/Status/TxPDO State
//     PlcTask Inputs/GVL_iXlinker.EtherCAT_Master_EPPxxxx.Beckhoff_EPP3xxx.Beckhoff_EPP3xxxEK1122.A_0002_EPP3174_0002_0017.AI_Standard_Channel_3.Status/TxPDO_State <-> AI Standard Channel 3/Status/TxPDO State
//     PlcTask Inputs/GVL_iXlinker.EtherCAT_Master_EPPxxxx.Beckhoff_EPP3xxx.Beckhoff_EPP3xxxEK1122.A_0002_EPP3174_0002_0017.AI_Standard_Channel_4.Status/TxPDO_State <-> AI Standard Channel 4/Status/TxPDO State
//     PlcTask Inputs/GVL_iXlinker.EtherCAT_Master_EPPxxxx.Beckhoff_EPP3xxx.Beckhoff_EPP3xxxEK1122.A_0002_EPP3174_0002_0017.AI_Standard_Channel_1.Status/TxPDO_Toggle <-> AI Standard Channel 1/Status/TxPDO Toggle
//     PlcTask Inputs/GVL_iXlinker.EtherCAT_Master_EPPxxxx.Beckhoff_EPP3xxx.Beckhoff_EPP3xxxEK1122.A_0002_EPP3174_0002_0017.AI_Standard_Channel_2.Status/TxPDO_Toggle <-> AI Standard Channel 2/Status/TxPDO Toggle
//     PlcTask Inputs/GVL_iXlinker.EtherCAT_Master_EPPxxxx.Beckhoff_EPP3xxx.Beckhoff_EPP3xxxEK1122.A_0002_EPP3174_0002_0017.AI_Standard_Channel_3.Status/TxPDO_Toggle <-> AI Standard Channel 3/Status/TxPDO Toggle
//     PlcTask Inputs/GVL_iXlinker.EtherCAT_Master_EPPxxxx.Beckhoff_EPP3xxx.Beckhoff_EPP3xxxEK1122.A_0002_EPP3174_0002_0017.AI_Standard_Channel_4.Status/TxPDO_Toggle <-> AI Standard Channel 4/Status/TxPDO Toggle
//     PlcTask Inputs/GVL_iXlinker.EtherCAT_Master_EPPxxxx.Beckhoff_EPP3xxx.Beckhoff_EPP3xxxEK1122.A_0002_EPP3174_0002_0017.AI_Standard_Channel_1.Value <-> AI Standard Channel 1/Value
//     PlcTask Inputs/GVL_iXlinker.EtherCAT_Master_EPPxxxx.Beckhoff_EPP3xxx.Beckhoff_EPP3xxxEK1122.A_0002_EPP3174_0002_0017.AI_Standard_Channel_2.Value <-> AI Standard Channel 2/Value
//     PlcTask Inputs/GVL_iXlinker.EtherCAT_Master_EPPxxxx.Beckhoff_EPP3xxx.Beckhoff_EPP3xxxEK1122.A_0002_EPP3174_0002_0017.AI_Standard_Channel_3.Value <-> AI Standard Channel 3/Value
//     PlcTask Inputs/GVL_iXlinker.EtherCAT_Master_EPPxxxx.Beckhoff_EPP3xxx.Beckhoff_EPP3xxxEK1122.A_0002_EPP3174_0002_0017.AI_Standard_Channel_4.Value <-> AI Standard Channel 4/Value
//     PlcTask Inputs/GVL_iXlinker.EtherCAT_Master_EPPxxxx.Beckhoff_EPP3xxx.Beckhoff_EPP3xxxEK1122.A_0002_EPP3174_0002_0017.WcState.WcState <-> WcState/WcState
//     PlcTask Inputs/GVL_iXlinker.EtherCAT_Master_EPPxxxx.Beckhoff_EPP3xxx.Beckhoff_EPP3xxxEK1122.A_0002_EPP3174_0002_0017.WcState.InputToggle <-> WcState/InputToggle
//     PlcTask Inputs/GVL_iXlinker.EtherCAT_Master_EPPxxxx.Beckhoff_EPP3xxx.Beckhoff_EPP3xxxEK1122.A_0002_EPP3174_0002_0017.InfoData.AdsAddr <-> InfoData/AdsAddr
//     PlcTask Inputs/GVL_iXlinker.EtherCAT_Master_EPPxxxx.Beckhoff_EPP3xxx.Beckhoff_EPP3xxxEK1122.A_0002_EPP3174_0002_0017.InfoData.State <-> InfoData/State
//   PLC/PLC Instance <-> EtherCAT Master EPPxxxx/Beckhoff EPP3xxx/Beckhoff EPP3xxxEK1122/A_0003(EPP3174-0002-0018)
//     PlcTask Inputs/GVL_iXlinker.EtherCAT_Master_EPPxxxx.Beckhoff_EPP3xxx.Beckhoff_EPP3xxxEK1122.A_0003_EPP3174_0002_0018.AI_Standard_Channel_1.Status/Underrange <-> AI Standard Channel 1/Status/Underrange
//     PlcTask Inputs/GVL_iXlinker.EtherCAT_Master_EPPxxxx.Beckhoff_EPP3xxx.Beckhoff_EPP3xxxEK1122.A_0003_EPP3174_0002_0018.AI_Standard_Channel_2.Status/Underrange <-> AI Standard Channel 2/Status/Underrange
//     PlcTask Inputs/GVL_iXlinker.EtherCAT_Master_EPPxxxx.Beckhoff_EPP3xxx.Beckhoff_EPP3xxxEK1122.A_0003_EPP3174_0002_0018.AI_Standard_Channel_3.Status/Underrange <-> AI Standard Channel 3/Status/Underrange
//     PlcTask Inputs/GVL_iXlinker.EtherCAT_Master_EPPxxxx.Beckhoff_EPP3xxx.Beckhoff_EPP3xxxEK1122.A_0003_EPP3174_0002_0018.AI_Standard_Channel_4.Status/Underrange <-> AI Standard Channel 4/Status/Underrange
//     PlcTask Inputs/GVL_iXlinker.EtherCAT_Master_EPPxxxx.Beckhoff_EPP3xxx.Beckhoff_EPP3xxxEK1122.A_0003_EPP3174_0002_0018.AI_Standard_Channel_1.Status/Overrange <-> AI Standard Channel 1/Status/Overrange
//     PlcTask Inputs/GVL_iXlinker.EtherCAT_Master_EPPxxxx.Beckhoff_EPP3xxx.Beckhoff_EPP3xxxEK1122.A_0003_EPP3174_0002_0018.AI_Standard_Channel_2.Status/Overrange <-> AI Standard Channel 2/Status/Overrange
//     PlcTask Inputs/GVL_iXlinker.EtherCAT_Master_EPPxxxx.Beckhoff_EPP3xxx.Beckhoff_EPP3xxxEK1122.A_0003_EPP3174_0002_0018.AI_Standard_Channel_3.Status/Overrange <-> AI Standard Channel 3/Status/Overrange
//     PlcTask Inputs/GVL_iXlinker.EtherCAT_Master_EPPxxxx.Beckhoff_EPP3xxx.Beckhoff_EPP3xxxEK1122.A_0003_EPP3174_0002_0018.AI_Standard_Channel_4.Status/Overrange <-> AI Standard Channel 4/Status/Overrange
//     PlcTask Inputs/GVL_iXlinker.EtherCAT_Master_EPPxxxx.Beckhoff_EPP3xxx.Beckhoff_EPP3xxxEK1122.A_0003_EPP3174_0002_0018.AI_Standard_Channel_1.Status/Limit_1 <-> AI Standard Channel 1/Status/Limit 1
//     PlcTask Inputs/GVL_iXlinker.EtherCAT_Master_EPPxxxx.Beckhoff_EPP3xxx.Beckhoff_EPP3xxxEK1122.A_0003_EPP3174_0002_0018.AI_Standard_Channel_1.Status/Limit_2 <-> AI Standard Channel 1/Status/Limit 2
//     PlcTask Inputs/GVL_iXlinker.EtherCAT_Master_EPPxxxx.Beckhoff_EPP3xxx.Beckhoff_EPP3xxxEK1122.A_0003_EPP3174_0002_0018.AI_Standard_Channel_2.Status/Limit_1 <-> AI Standard Channel 2/Status/Limit 1
//     PlcTask Inputs/GVL_iXlinker.EtherCAT_Master_EPPxxxx.Beckhoff_EPP3xxx.Beckhoff_EPP3xxxEK1122.A_0003_EPP3174_0002_0018.AI_Standard_Channel_2.Status/Limit_2 <-> AI Standard Channel 2/Status/Limit 2
//     PlcTask Inputs/GVL_iXlinker.EtherCAT_Master_EPPxxxx.Beckhoff_EPP3xxx.Beckhoff_EPP3xxxEK1122.A_0003_EPP3174_0002_0018.AI_Standard_Channel_3.Status/Limit_1 <-> AI Standard Channel 3/Status/Limit 1
//     PlcTask Inputs/GVL_iXlinker.EtherCAT_Master_EPPxxxx.Beckhoff_EPP3xxx.Beckhoff_EPP3xxxEK1122.A_0003_EPP3174_0002_0018.AI_Standard_Channel_3.Status/Limit_2 <-> AI Standard Channel 3/Status/Limit 2
//     PlcTask Inputs/GVL_iXlinker.EtherCAT_Master_EPPxxxx.Beckhoff_EPP3xxx.Beckhoff_EPP3xxxEK1122.A_0003_EPP3174_0002_0018.AI_Standard_Channel_4.Status/Limit_1 <-> AI Standard Channel 4/Status/Limit 1
//     PlcTask Inputs/GVL_iXlinker.EtherCAT_Master_EPPxxxx.Beckhoff_EPP3xxx.Beckhoff_EPP3xxxEK1122.A_0003_EPP3174_0002_0018.AI_Standard_Channel_4.Status/Limit_2 <-> AI Standard Channel 4/Status/Limit 2
//     PlcTask Inputs/GVL_iXlinker.EtherCAT_Master_EPPxxxx.Beckhoff_EPP3xxx.Beckhoff_EPP3xxxEK1122.A_0003_EPP3174_0002_0018.AI_Standard_Channel_1.Status/Error <-> AI Standard Channel 1/Status/Error
//     PlcTask Inputs/GVL_iXlinker.EtherCAT_Master_EPPxxxx.Beckhoff_EPP3xxx.Beckhoff_EPP3xxxEK1122.A_0003_EPP3174_0002_0018.AI_Standard_Channel_2.Status/Error <-> AI Standard Channel 2/Status/Error
//     PlcTask Inputs/GVL_iXlinker.EtherCAT_Master_EPPxxxx.Beckhoff_EPP3xxx.Beckhoff_EPP3xxxEK1122.A_0003_EPP3174_0002_0018.AI_Standard_Channel_3.Status/Error <-> AI Standard Channel 3/Status/Error
//     PlcTask Inputs/GVL_iXlinker.EtherCAT_Master_EPPxxxx.Beckhoff_EPP3xxx.Beckhoff_EPP3xxxEK1122.A_0003_EPP3174_0002_0018.AI_Standard_Channel_4.Status/Error <-> AI Standard Channel 4/Status/Error
//     PlcTask Inputs/GVL_iXlinker.EtherCAT_Master_EPPxxxx.Beckhoff_EPP3xxx.Beckhoff_EPP3xxxEK1122.A_0003_EPP3174_0002_0018.AI_Standard_Channel_1.Status/Sync_error <-> AI Standard Channel 1/Status/Sync error
//     PlcTask Inputs/GVL_iXlinker.EtherCAT_Master_EPPxxxx.Beckhoff_EPP3xxx.Beckhoff_EPP3xxxEK1122.A_0003_EPP3174_0002_0018.AI_Standard_Channel_2.Status/Sync_error <-> AI Standard Channel 2/Status/Sync error
//     PlcTask Inputs/GVL_iXlinker.EtherCAT_Master_EPPxxxx.Beckhoff_EPP3xxx.Beckhoff_EPP3xxxEK1122.A_0003_EPP3174_0002_0018.AI_Standard_Channel_3.Status/Sync_error <-> AI Standard Channel 3/Status/Sync error
//     PlcTask Inputs/GVL_iXlinker.EtherCAT_Master_EPPxxxx.Beckhoff_EPP3xxx.Beckhoff_EPP3xxxEK1122.A_0003_EPP3174_0002_0018.AI_Standard_Channel_4.Status/Sync_error <-> AI Standard Channel 4/Status/Sync error
//     PlcTask Inputs/GVL_iXlinker.EtherCAT_Master_EPPxxxx.Beckhoff_EPP3xxx.Beckhoff_EPP3xxxEK1122.A_0003_EPP3174_0002_0018.AI_Standard_Channel_1.Status/TxPDO_State <-> AI Standard Channel 1/Status/TxPDO State
//     PlcTask Inputs/GVL_iXlinker.EtherCAT_Master_EPPxxxx.Beckhoff_EPP3xxx.Beckhoff_EPP3xxxEK1122.A_0003_EPP3174_0002_0018.AI_Standard_Channel_2.Status/TxPDO_State <-> AI Standard Channel 2/Status/TxPDO State
//     PlcTask Inputs/GVL_iXlinker.EtherCAT_Master_EPPxxxx.Beckhoff_EPP3xxx.Beckhoff_EPP3xxxEK1122.A_0003_EPP3174_0002_0018.AI_Standard_Channel_3.Status/TxPDO_State <-> AI Standard Channel 3/Status/TxPDO State
//     PlcTask Inputs/GVL_iXlinker.EtherCAT_Master_EPPxxxx.Beckhoff_EPP3xxx.Beckhoff_EPP3xxxEK1122.A_0003_EPP3174_0002_0018.AI_Standard_Channel_4.Status/TxPDO_State <-> AI Standard Channel 4/Status/TxPDO State
//     PlcTask Inputs/GVL_iXlinker.EtherCAT_Master_EPPxxxx.Beckhoff_EPP3xxx.Beckhoff_EPP3xxxEK1122.A_0003_EPP3174_0002_0018.AI_Standard_Channel_1.Status/TxPDO_Toggle <-> AI Standard Channel 1/Status/TxPDO Toggle
//     PlcTask Inputs/GVL_iXlinker.EtherCAT_Master_EPPxxxx.Beckhoff_EPP3xxx.Beckhoff_EPP3xxxEK1122.A_0003_EPP3174_0002_0018.AI_Standard_Channel_2.Status/TxPDO_Toggle <-> AI Standard Channel 2/Status/TxPDO Toggle
//     PlcTask Inputs/GVL_iXlinker.EtherCAT_Master_EPPxxxx.Beckhoff_EPP3xxx.Beckhoff_EPP3xxxEK1122.A_0003_EPP3174_0002_0018.AI_Standard_Channel_3.Status/TxPDO_Toggle <-> AI Standard Channel 3/Status/TxPDO Toggle
//     PlcTask Inputs/GVL_iXlinker.EtherCAT_Master_EPPxxxx.Beckhoff_EPP3xxx.Beckhoff_EPP3xxxEK1122.A_0003_EPP3174_0002_0018.AI_Standard_Channel_4.Status/TxPDO_Toggle <-> AI Standard Channel 4/Status/TxPDO Toggle
//     PlcTask Inputs/GVL_iXlinker.EtherCAT_Master_EPPxxxx.Beckhoff_EPP3xxx.Beckhoff_EPP3xxxEK1122.A_0003_EPP3174_0002_0018.AI_Standard_Channel_1.Value <-> AI Standard Channel 1/Value
//     PlcTask Inputs/GVL_iXlinker.EtherCAT_Master_EPPxxxx.Beckhoff_EPP3xxx.Beckhoff_EPP3xxxEK1122.A_0003_EPP3174_0002_0018.AI_Standard_Channel_2.Value <-> AI Standard Channel 2/Value
//     PlcTask Inputs/GVL_iXlinker.EtherCAT_Master_EPPxxxx.Beckhoff_EPP3xxx.Beckhoff_EPP3xxxEK1122.A_0003_EPP3174_0002_0018.AI_Standard_Channel_3.Value <-> AI Standard Channel 3/Value
//     PlcTask Inputs/GVL_iXlinker.EtherCAT_Master_EPPxxxx.Beckhoff_EPP3xxx.Beckhoff_EPP3xxxEK1122.A_0003_EPP3174_0002_0018.AI_Standard_Channel_4.Value <-> AI Standard Channel 4/Value
//     PlcTask Inputs/GVL_iXlinker.EtherCAT_Master_EPPxxxx.Beckhoff_EPP3xxx.Beckhoff_EPP3xxxEK1122.A_0003_EPP3174_0002_0018.WcState.WcState <-> WcState/WcState
//     PlcTask Inputs/GVL_iXlinker.EtherCAT_Master_EPPxxxx.Beckhoff_EPP3xxx.Beckhoff_EPP3xxxEK1122.A_0003_EPP3174_0002_0018.WcState.InputToggle <-> WcState/InputToggle
//     PlcTask Inputs/GVL_iXlinker.EtherCAT_Master_EPPxxxx.Beckhoff_EPP3xxx.Beckhoff_EPP3xxxEK1122.A_0003_EPP3174_0002_0018.InfoData.AdsAddr <-> InfoData/AdsAddr
//     PlcTask Inputs/GVL_iXlinker.EtherCAT_Master_EPPxxxx.Beckhoff_EPP3xxx.Beckhoff_EPP3xxxEK1122.A_0003_EPP3174_0002_0018.InfoData.State <-> InfoData/State
//   PLC/PLC Instance <-> EtherCAT Master EPPxxxx/Beckhoff EPP3xxx/Beckhoff EPP3xxxEK1122/A_0004(EPP3184-0002-0016)
//     PlcTask Inputs/GVL_iXlinker.EtherCAT_Master_EPPxxxx.Beckhoff_EPP3xxx.Beckhoff_EPP3xxxEK1122.A_0004_EPP3184_0002_0016.AI_Standard_Channel_1.Status/Underrange <-> AI Standard Channel 1/Status/Underrange
//     PlcTask Inputs/GVL_iXlinker.EtherCAT_Master_EPPxxxx.Beckhoff_EPP3xxx.Beckhoff_EPP3xxxEK1122.A_0004_EPP3184_0002_0016.AI_Standard_Channel_2.Status/Underrange <-> AI Standard Channel 2/Status/Underrange
//     PlcTask Inputs/GVL_iXlinker.EtherCAT_Master_EPPxxxx.Beckhoff_EPP3xxx.Beckhoff_EPP3xxxEK1122.A_0004_EPP3184_0002_0016.AI_Standard_Channel_3.Status/Underrange <-> AI Standard Channel 3/Status/Underrange
//     PlcTask Inputs/GVL_iXlinker.EtherCAT_Master_EPPxxxx.Beckhoff_EPP3xxx.Beckhoff_EPP3xxxEK1122.A_0004_EPP3184_0002_0016.AI_Standard_Channel_4.Status/Underrange <-> AI Standard Channel 4/Status/Underrange
//     PlcTask Inputs/GVL_iXlinker.EtherCAT_Master_EPPxxxx.Beckhoff_EPP3xxx.Beckhoff_EPP3xxxEK1122.A_0004_EPP3184_0002_0016.AI_Standard_Channel_1.Status/Overrange <-> AI Standard Channel 1/Status/Overrange
//     PlcTask Inputs/GVL_iXlinker.EtherCAT_Master_EPPxxxx.Beckhoff_EPP3xxx.Beckhoff_EPP3xxxEK1122.A_0004_EPP3184_0002_0016.AI_Standard_Channel_2.Status/Overrange <-> AI Standard Channel 2/Status/Overrange
//     PlcTask Inputs/GVL_iXlinker.EtherCAT_Master_EPPxxxx.Beckhoff_EPP3xxx.Beckhoff_EPP3xxxEK1122.A_0004_EPP3184_0002_0016.AI_Standard_Channel_3.Status/Overrange <-> AI Standard Channel 3/Status/Overrange
//     PlcTask Inputs/GVL_iXlinker.EtherCAT_Master_EPPxxxx.Beckhoff_EPP3xxx.Beckhoff_EPP3xxxEK1122.A_0004_EPP3184_0002_0016.AI_Standard_Channel_4.Status/Overrange <-> AI Standard Channel 4/Status/Overrange
//     PlcTask Inputs/GVL_iXlinker.EtherCAT_Master_EPPxxxx.Beckhoff_EPP3xxx.Beckhoff_EPP3xxxEK1122.A_0004_EPP3184_0002_0016.AI_Standard_Channel_1.Status/Limit_1 <-> AI Standard Channel 1/Status/Limit 1
//     PlcTask Inputs/GVL_iXlinker.EtherCAT_Master_EPPxxxx.Beckhoff_EPP3xxx.Beckhoff_EPP3xxxEK1122.A_0004_EPP3184_0002_0016.AI_Standard_Channel_1.Status/Limit_2 <-> AI Standard Channel 1/Status/Limit 2
//     PlcTask Inputs/GVL_iXlinker.EtherCAT_Master_EPPxxxx.Beckhoff_EPP3xxx.Beckhoff_EPP3xxxEK1122.A_0004_EPP3184_0002_0016.AI_Standard_Channel_2.Status/Limit_1 <-> AI Standard Channel 2/Status/Limit 1
//     PlcTask Inputs/GVL_iXlinker.EtherCAT_Master_EPPxxxx.Beckhoff_EPP3xxx.Beckhoff_EPP3xxxEK1122.A_0004_EPP3184_0002_0016.AI_Standard_Channel_2.Status/Limit_2 <-> AI Standard Channel 2/Status/Limit 2
//     PlcTask Inputs/GVL_iXlinker.EtherCAT_Master_EPPxxxx.Beckhoff_EPP3xxx.Beckhoff_EPP3xxxEK1122.A_0004_EPP3184_0002_0016.AI_Standard_Channel_3.Status/Limit_1 <-> AI Standard Channel 3/Status/Limit 1
//     PlcTask Inputs/GVL_iXlinker.EtherCAT_Master_EPPxxxx.Beckhoff_EPP3xxx.Beckhoff_EPP3xxxEK1122.A_0004_EPP3184_0002_0016.AI_Standard_Channel_3.Status/Limit_2 <-> AI Standard Channel 3/Status/Limit 2
//     PlcTask Inputs/GVL_iXlinker.EtherCAT_Master_EPPxxxx.Beckhoff_EPP3xxx.Beckhoff_EPP3xxxEK1122.A_0004_EPP3184_0002_0016.AI_Standard_Channel_4.Status/Limit_1 <-> AI Standard Channel 4/Status/Limit 1
//     PlcTask Inputs/GVL_iXlinker.EtherCAT_Master_EPPxxxx.Beckhoff_EPP3xxx.Beckhoff_EPP3xxxEK1122.A_0004_EPP3184_0002_0016.AI_Standard_Channel_4.Status/Limit_2 <-> AI Standard Channel 4/Status/Limit 2
//     PlcTask Inputs/GVL_iXlinker.EtherCAT_Master_EPPxxxx.Beckhoff_EPP3xxx.Beckhoff_EPP3xxxEK1122.A_0004_EPP3184_0002_0016.AI_Standard_Channel_1.Status/Error <-> AI Standard Channel 1/Status/Error
//     PlcTask Inputs/GVL_iXlinker.EtherCAT_Master_EPPxxxx.Beckhoff_EPP3xxx.Beckhoff_EPP3xxxEK1122.A_0004_EPP3184_0002_0016.AI_Standard_Channel_2.Status/Error <-> AI Standard Channel 2/Status/Error
//     PlcTask Inputs/GVL_iXlinker.EtherCAT_Master_EPPxxxx.Beckhoff_EPP3xxx.Beckhoff_EPP3xxxEK1122.A_0004_EPP3184_0002_0016.AI_Standard_Channel_3.Status/Error <-> AI Standard Channel 3/Status/Error
//     PlcTask Inputs/GVL_iXlinker.EtherCAT_Master_EPPxxxx.Beckhoff_EPP3xxx.Beckhoff_EPP3xxxEK1122.A_0004_EPP3184_0002_0016.AI_Standard_Channel_4.Status/Error <-> AI Standard Channel 4/Status/Error
//     PlcTask Inputs/GVL_iXlinker.EtherCAT_Master_EPPxxxx.Beckhoff_EPP3xxx.Beckhoff_EPP3xxxEK1122.A_0004_EPP3184_0002_0016.AI_Standard_Channel_1.Status/Sync_error <-> AI Standard Channel 1/Status/Sync error
//     PlcTask Inputs/GVL_iXlinker.EtherCAT_Master_EPPxxxx.Beckhoff_EPP3xxx.Beckhoff_EPP3xxxEK1122.A_0004_EPP3184_0002_0016.AI_Standard_Channel_2.Status/Sync_error <-> AI Standard Channel 2/Status/Sync error
//     PlcTask Inputs/GVL_iXlinker.EtherCAT_Master_EPPxxxx.Beckhoff_EPP3xxx.Beckhoff_EPP3xxxEK1122.A_0004_EPP3184_0002_0016.AI_Standard_Channel_3.Status/Sync_error <-> AI Standard Channel 3/Status/Sync error
//     PlcTask Inputs/GVL_iXlinker.EtherCAT_Master_EPPxxxx.Beckhoff_EPP3xxx.Beckhoff_EPP3xxxEK1122.A_0004_EPP3184_0002_0016.AI_Standard_Channel_4.Status/Sync_error <-> AI Standard Channel 4/Status/Sync error
//     PlcTask Inputs/GVL_iXlinker.EtherCAT_Master_EPPxxxx.Beckhoff_EPP3xxx.Beckhoff_EPP3xxxEK1122.A_0004_EPP3184_0002_0016.AI_Standard_Channel_1.Status/TxPDO_State <-> AI Standard Channel 1/Status/TxPDO State
//     PlcTask Inputs/GVL_iXlinker.EtherCAT_Master_EPPxxxx.Beckhoff_EPP3xxx.Beckhoff_EPP3xxxEK1122.A_0004_EPP3184_0002_0016.AI_Standard_Channel_2.Status/TxPDO_State <-> AI Standard Channel 2/Status/TxPDO State
//     PlcTask Inputs/GVL_iXlinker.EtherCAT_Master_EPPxxxx.Beckhoff_EPP3xxx.Beckhoff_EPP3xxxEK1122.A_0004_EPP3184_0002_0016.AI_Standard_Channel_3.Status/TxPDO_State <-> AI Standard Channel 3/Status/TxPDO State
//     PlcTask Inputs/GVL_iXlinker.EtherCAT_Master_EPPxxxx.Beckhoff_EPP3xxx.Beckhoff_EPP3xxxEK1122.A_0004_EPP3184_0002_0016.AI_Standard_Channel_4.Status/TxPDO_State <-> AI Standard Channel 4/Status/TxPDO State
//     PlcTask Inputs/GVL_iXlinker.EtherCAT_Master_EPPxxxx.Beckhoff_EPP3xxx.Beckhoff_EPP3xxxEK1122.A_0004_EPP3184_0002_0016.AI_Standard_Channel_1.Status/TxPDO_Toggle <-> AI Standard Channel 1/Status/TxPDO Toggle
//     PlcTask Inputs/GVL_iXlinker.EtherCAT_Master_EPPxxxx.Beckhoff_EPP3xxx.Beckhoff_EPP3xxxEK1122.A_0004_EPP3184_0002_0016.AI_Standard_Channel_2.Status/TxPDO_Toggle <-> AI Standard Channel 2/Status/TxPDO Toggle
//     PlcTask Inputs/GVL_iXlinker.EtherCAT_Master_EPPxxxx.Beckhoff_EPP3xxx.Beckhoff_EPP3xxxEK1122.A_0004_EPP3184_0002_0016.AI_Standard_Channel_3.Status/TxPDO_Toggle <-> AI Standard Channel 3/Status/TxPDO Toggle
//     PlcTask Inputs/GVL_iXlinker.EtherCAT_Master_EPPxxxx.Beckhoff_EPP3xxx.Beckhoff_EPP3xxxEK1122.A_0004_EPP3184_0002_0016.AI_Standard_Channel_4.Status/TxPDO_Toggle <-> AI Standard Channel 4/Status/TxPDO Toggle
//     PlcTask Inputs/GVL_iXlinker.EtherCAT_Master_EPPxxxx.Beckhoff_EPP3xxx.Beckhoff_EPP3xxxEK1122.A_0004_EPP3184_0002_0016.AI_Standard_Channel_1.Value <-> AI Standard Channel 1/Value
//     PlcTask Inputs/GVL_iXlinker.EtherCAT_Master_EPPxxxx.Beckhoff_EPP3xxx.Beckhoff_EPP3xxxEK1122.A_0004_EPP3184_0002_0016.AI_Standard_Channel_2.Value <-> AI Standard Channel 2/Value
//     PlcTask Inputs/GVL_iXlinker.EtherCAT_Master_EPPxxxx.Beckhoff_EPP3xxx.Beckhoff_EPP3xxxEK1122.A_0004_EPP3184_0002_0016.AI_Standard_Channel_3.Value <-> AI Standard Channel 3/Value
//     PlcTask Inputs/GVL_iXlinker.EtherCAT_Master_EPPxxxx.Beckhoff_EPP3xxx.Beckhoff_EPP3xxxEK1122.A_0004_EPP3184_0002_0016.AI_Standard_Channel_4.Value <-> AI Standard Channel 4/Value
//     PlcTask Inputs/GVL_iXlinker.EtherCAT_Master_EPPxxxx.Beckhoff_EPP3xxx.Beckhoff_EPP3xxxEK1122.A_0004_EPP3184_0002_0016.WcState.WcState <-> WcState/WcState
//     PlcTask Inputs/GVL_iXlinker.EtherCAT_Master_EPPxxxx.Beckhoff_EPP3xxx.Beckhoff_EPP3xxxEK1122.A_0004_EPP3184_0002_0016.WcState.InputToggle <-> WcState/InputToggle
//     PlcTask Inputs/GVL_iXlinker.EtherCAT_Master_EPPxxxx.Beckhoff_EPP3xxx.Beckhoff_EPP3xxxEK1122.A_0004_EPP3184_0002_0016.InfoData.AdsAddr <-> InfoData/AdsAddr
//     PlcTask Inputs/GVL_iXlinker.EtherCAT_Master_EPPxxxx.Beckhoff_EPP3xxx.Beckhoff_EPP3xxxEK1122.A_0004_EPP3184_0002_0016.InfoData.State <-> InfoData/State
//   PLC/PLC Instance <-> EtherCAT Master EPPxxxx/Beckhoff EPP3xxx/Beckhoff EPP3xxxEK1122/A_0005(EPP3184-0002-0017)
//     PlcTask Inputs/GVL_iXlinker.EtherCAT_Master_EPPxxxx.Beckhoff_EPP3xxx.Beckhoff_EPP3xxxEK1122.A_0005_EPP3184_0002_0017.AI_Standard_Channel_1.Status/Underrange <-> AI Standard Channel 1/Status/Underrange
//     PlcTask Inputs/GVL_iXlinker.EtherCAT_Master_EPPxxxx.Beckhoff_EPP3xxx.Beckhoff_EPP3xxxEK1122.A_0005_EPP3184_0002_0017.AI_Standard_Channel_2.Status/Underrange <-> AI Standard Channel 2/Status/Underrange
//     PlcTask Inputs/GVL_iXlinker.EtherCAT_Master_EPPxxxx.Beckhoff_EPP3xxx.Beckhoff_EPP3xxxEK1122.A_0005_EPP3184_0002_0017.AI_Standard_Channel_3.Status/Underrange <-> AI Standard Channel 3/Status/Underrange
//     PlcTask Inputs/GVL_iXlinker.EtherCAT_Master_EPPxxxx.Beckhoff_EPP3xxx.Beckhoff_EPP3xxxEK1122.A_0005_EPP3184_0002_0017.AI_Standard_Channel_4.Status/Underrange <-> AI Standard Channel 4/Status/Underrange
//     PlcTask Inputs/GVL_iXlinker.EtherCAT_Master_EPPxxxx.Beckhoff_EPP3xxx.Beckhoff_EPP3xxxEK1122.A_0005_EPP3184_0002_0017.AI_Standard_Channel_1.Status/Overrange <-> AI Standard Channel 1/Status/Overrange
//     PlcTask Inputs/GVL_iXlinker.EtherCAT_Master_EPPxxxx.Beckhoff_EPP3xxx.Beckhoff_EPP3xxxEK1122.A_0005_EPP3184_0002_0017.AI_Standard_Channel_2.Status/Overrange <-> AI Standard Channel 2/Status/Overrange
//     PlcTask Inputs/GVL_iXlinker.EtherCAT_Master_EPPxxxx.Beckhoff_EPP3xxx.Beckhoff_EPP3xxxEK1122.A_0005_EPP3184_0002_0017.AI_Standard_Channel_3.Status/Overrange <-> AI Standard Channel 3/Status/Overrange
//     PlcTask Inputs/GVL_iXlinker.EtherCAT_Master_EPPxxxx.Beckhoff_EPP3xxx.Beckhoff_EPP3xxxEK1122.A_0005_EPP3184_0002_0017.AI_Standard_Channel_4.Status/Overrange <-> AI Standard Channel 4/Status/Overrange
//     PlcTask Inputs/GVL_iXlinker.EtherCAT_Master_EPPxxxx.Beckhoff_EPP3xxx.Beckhoff_EPP3xxxEK1122.A_0005_EPP3184_0002_0017.AI_Standard_Channel_1.Status/Limit_1 <-> AI Standard Channel 1/Status/Limit 1
//     PlcTask Inputs/GVL_iXlinker.EtherCAT_Master_EPPxxxx.Beckhoff_EPP3xxx.Beckhoff_EPP3xxxEK1122.A_0005_EPP3184_0002_0017.AI_Standard_Channel_1.Status/Limit_2 <-> AI Standard Channel 1/Status/Limit 2
//     PlcTask Inputs/GVL_iXlinker.EtherCAT_Master_EPPxxxx.Beckhoff_EPP3xxx.Beckhoff_EPP3xxxEK1122.A_0005_EPP3184_0002_0017.AI_Standard_Channel_2.Status/Limit_1 <-> AI Standard Channel 2/Status/Limit 1
//     PlcTask Inputs/GVL_iXlinker.EtherCAT_Master_EPPxxxx.Beckhoff_EPP3xxx.Beckhoff_EPP3xxxEK1122.A_0005_EPP3184_0002_0017.AI_Standard_Channel_2.Status/Limit_2 <-> AI Standard Channel 2/Status/Limit 2
//     PlcTask Inputs/GVL_iXlinker.EtherCAT_Master_EPPxxxx.Beckhoff_EPP3xxx.Beckhoff_EPP3xxxEK1122.A_0005_EPP3184_0002_0017.AI_Standard_Channel_3.Status/Limit_1 <-> AI Standard Channel 3/Status/Limit 1
//     PlcTask Inputs/GVL_iXlinker.EtherCAT_Master_EPPxxxx.Beckhoff_EPP3xxx.Beckhoff_EPP3xxxEK1122.A_0005_EPP3184_0002_0017.AI_Standard_Channel_3.Status/Limit_2 <-> AI Standard Channel 3/Status/Limit 2
//     PlcTask Inputs/GVL_iXlinker.EtherCAT_Master_EPPxxxx.Beckhoff_EPP3xxx.Beckhoff_EPP3xxxEK1122.A_0005_EPP3184_0002_0017.AI_Standard_Channel_4.Status/Limit_1 <-> AI Standard Channel 4/Status/Limit 1
//     PlcTask Inputs/GVL_iXlinker.EtherCAT_Master_EPPxxxx.Beckhoff_EPP3xxx.Beckhoff_EPP3xxxEK1122.A_0005_EPP3184_0002_0017.AI_Standard_Channel_4.Status/Limit_2 <-> AI Standard Channel 4/Status/Limit 2
//     PlcTask Inputs/GVL_iXlinker.EtherCAT_Master_EPPxxxx.Beckhoff_EPP3xxx.Beckhoff_EPP3xxxEK1122.A_0005_EPP3184_0002_0017.AI_Standard_Channel_1.Status/Error <-> AI Standard Channel 1/Status/Error
//     PlcTask Inputs/GVL_iXlinker.EtherCAT_Master_EPPxxxx.Beckhoff_EPP3xxx.Beckhoff_EPP3xxxEK1122.A_0005_EPP3184_0002_0017.AI_Standard_Channel_2.Status/Error <-> AI Standard Channel 2/Status/Error
//     PlcTask Inputs/GVL_iXlinker.EtherCAT_Master_EPPxxxx.Beckhoff_EPP3xxx.Beckhoff_EPP3xxxEK1122.A_0005_EPP3184_0002_0017.AI_Standard_Channel_3.Status/Error <-> AI Standard Channel 3/Status/Error
//     PlcTask Inputs/GVL_iXlinker.EtherCAT_Master_EPPxxxx.Beckhoff_EPP3xxx.Beckhoff_EPP3xxxEK1122.A_0005_EPP3184_0002_0017.AI_Standard_Channel_4.Status/Error <-> AI Standard Channel 4/Status/Error
//     PlcTask Inputs/GVL_iXlinker.EtherCAT_Master_EPPxxxx.Beckhoff_EPP3xxx.Beckhoff_EPP3xxxEK1122.A_0005_EPP3184_0002_0017.AI_Standard_Channel_1.Status/Sync_error <-> AI Standard Channel 1/Status/Sync error
//     PlcTask Inputs/GVL_iXlinker.EtherCAT_Master_EPPxxxx.Beckhoff_EPP3xxx.Beckhoff_EPP3xxxEK1122.A_0005_EPP3184_0002_0017.AI_Standard_Channel_2.Status/Sync_error <-> AI Standard Channel 2/Status/Sync error
//     PlcTask Inputs/GVL_iXlinker.EtherCAT_Master_EPPxxxx.Beckhoff_EPP3xxx.Beckhoff_EPP3xxxEK1122.A_0005_EPP3184_0002_0017.AI_Standard_Channel_3.Status/Sync_error <-> AI Standard Channel 3/Status/Sync error
//     PlcTask Inputs/GVL_iXlinker.EtherCAT_Master_EPPxxxx.Beckhoff_EPP3xxx.Beckhoff_EPP3xxxEK1122.A_0005_EPP3184_0002_0017.AI_Standard_Channel_4.Status/Sync_error <-> AI Standard Channel 4/Status/Sync error
//     PlcTask Inputs/GVL_iXlinker.EtherCAT_Master_EPPxxxx.Beckhoff_EPP3xxx.Beckhoff_EPP3xxxEK1122.A_0005_EPP3184_0002_0017.AI_Standard_Channel_1.Status/TxPDO_State <-> AI Standard Channel 1/Status/TxPDO State
//     PlcTask Inputs/GVL_iXlinker.EtherCAT_Master_EPPxxxx.Beckhoff_EPP3xxx.Beckhoff_EPP3xxxEK1122.A_0005_EPP3184_0002_0017.AI_Standard_Channel_2.Status/TxPDO_State <-> AI Standard Channel 2/Status/TxPDO State
//     PlcTask Inputs/GVL_iXlinker.EtherCAT_Master_EPPxxxx.Beckhoff_EPP3xxx.Beckhoff_EPP3xxxEK1122.A_0005_EPP3184_0002_0017.AI_Standard_Channel_3.Status/TxPDO_State <-> AI Standard Channel 3/Status/TxPDO State
//     PlcTask Inputs/GVL_iXlinker.EtherCAT_Master_EPPxxxx.Beckhoff_EPP3xxx.Beckhoff_EPP3xxxEK1122.A_0005_EPP3184_0002_0017.AI_Standard_Channel_4.Status/TxPDO_State <-> AI Standard Channel 4/Status/TxPDO State
//     PlcTask Inputs/GVL_iXlinker.EtherCAT_Master_EPPxxxx.Beckhoff_EPP3xxx.Beckhoff_EPP3xxxEK1122.A_0005_EPP3184_0002_0017.AI_Standard_Channel_1.Status/TxPDO_Toggle <-> AI Standard Channel 1/Status/TxPDO Toggle
//     PlcTask Inputs/GVL_iXlinker.EtherCAT_Master_EPPxxxx.Beckhoff_EPP3xxx.Beckhoff_EPP3xxxEK1122.A_0005_EPP3184_0002_0017.AI_Standard_Channel_2.Status/TxPDO_Toggle <-> AI Standard Channel 2/Status/TxPDO Toggle
//     PlcTask Inputs/GVL_iXlinker.EtherCAT_Master_EPPxxxx.Beckhoff_EPP3xxx.Beckhoff_EPP3xxxEK1122.A_0005_EPP3184_0002_0017.AI_Standard_Channel_3.Status/TxPDO_Toggle <-> AI Standard Channel 3/Status/TxPDO Toggle
//     PlcTask Inputs/GVL_iXlinker.EtherCAT_Master_EPPxxxx.Beckhoff_EPP3xxx.Beckhoff_EPP3xxxEK1122.A_0005_EPP3184_0002_0017.AI_Standard_Channel_4.Status/TxPDO_Toggle <-> AI Standard Channel 4/Status/TxPDO Toggle
//     PlcTask Inputs/GVL_iXlinker.EtherCAT_Master_EPPxxxx.Beckhoff_EPP3xxx.Beckhoff_EPP3xxxEK1122.A_0005_EPP3184_0002_0017.AI_Standard_Channel_1.Value <-> AI Standard Channel 1/Value
//     PlcTask Inputs/GVL_iXlinker.EtherCAT_Master_EPPxxxx.Beckhoff_EPP3xxx.Beckhoff_EPP3xxxEK1122.A_0005_EPP3184_0002_0017.AI_Standard_Channel_2.Value <-> AI Standard Channel 2/Value
//     PlcTask Inputs/GVL_iXlinker.EtherCAT_Master_EPPxxxx.Beckhoff_EPP3xxx.Beckhoff_EPP3xxxEK1122.A_0005_EPP3184_0002_0017.AI_Standard_Channel_3.Value <-> AI Standard Channel 3/Value
//     PlcTask Inputs/GVL_iXlinker.EtherCAT_Master_EPPxxxx.Beckhoff_EPP3xxx.Beckhoff_EPP3xxxEK1122.A_0005_EPP3184_0002_0017.AI_Standard_Channel_4.Value <-> AI Standard Channel 4/Value
//     PlcTask Inputs/GVL_iXlinker.EtherCAT_Master_EPPxxxx.Beckhoff_EPP3xxx.Beckhoff_EPP3xxxEK1122.A_0005_EPP3184_0002_0017.WcState.WcState <-> WcState/WcState
//     PlcTask Inputs/GVL_iXlinker.EtherCAT_Master_EPPxxxx.Beckhoff_EPP3xxx.Beckhoff_EPP3xxxEK1122.A_0005_EPP3184_0002_0017.WcState.InputToggle <-> WcState/InputToggle
//     PlcTask Inputs/GVL_iXlinker.EtherCAT_Master_EPPxxxx.Beckhoff_EPP3xxx.Beckhoff_EPP3xxxEK1122.A_0005_EPP3184_0002_0017.InfoData.AdsAddr <-> InfoData/AdsAddr
//     PlcTask Inputs/GVL_iXlinker.EtherCAT_Master_EPPxxxx.Beckhoff_EPP3xxx.Beckhoff_EPP3xxxEK1122.A_0005_EPP3184_0002_0017.InfoData.State <-> InfoData/State
//   PLC/PLC Instance <-> EtherCAT Master EPPxxxx/Beckhoff EPP3xxx/Beckhoff EPP3xxxEK1122/A_0006(EPP3184-0002-0018)
//     PlcTask Inputs/GVL_iXlinker.EtherCAT_Master_EPPxxxx.Beckhoff_EPP3xxx.Beckhoff_EPP3xxxEK1122.A_0006_EPP3184_0002_0018.AI_Standard_Channel_1.Status/Underrange <-> AI Standard Channel 1/Status/Underrange
//     PlcTask Inputs/GVL_iXlinker.EtherCAT_Master_EPPxxxx.Beckhoff_EPP3xxx.Beckhoff_EPP3xxxEK1122.A_0006_EPP3184_0002_0018.AI_Standard_Channel_2.Status/Underrange <-> AI Standard Channel 2/Status/Underrange
//     PlcTask Inputs/GVL_iXlinker.EtherCAT_Master_EPPxxxx.Beckhoff_EPP3xxx.Beckhoff_EPP3xxxEK1122.A_0006_EPP3184_0002_0018.AI_Standard_Channel_3.Status/Underrange <-> AI Standard Channel 3/Status/Underrange
//     PlcTask Inputs/GVL_iXlinker.EtherCAT_Master_EPPxxxx.Beckhoff_EPP3xxx.Beckhoff_EPP3xxxEK1122.A_0006_EPP3184_0002_0018.AI_Standard_Channel_4.Status/Underrange <-> AI Standard Channel 4/Status/Underrange
//     PlcTask Inputs/GVL_iXlinker.EtherCAT_Master_EPPxxxx.Beckhoff_EPP3xxx.Beckhoff_EPP3xxxEK1122.A_0006_EPP3184_0002_0018.AI_Standard_Channel_1.Status/Overrange <-> AI Standard Channel 1/Status/Overrange
//     PlcTask Inputs/GVL_iXlinker.EtherCAT_Master_EPPxxxx.Beckhoff_EPP3xxx.Beckhoff_EPP3xxxEK1122.A_0006_EPP3184_0002_0018.AI_Standard_Channel_2.Status/Overrange <-> AI Standard Channel 2/Status/Overrange
//     PlcTask Inputs/GVL_iXlinker.EtherCAT_Master_EPPxxxx.Beckhoff_EPP3xxx.Beckhoff_EPP3xxxEK1122.A_0006_EPP3184_0002_0018.AI_Standard_Channel_3.Status/Overrange <-> AI Standard Channel 3/Status/Overrange
//     PlcTask Inputs/GVL_iXlinker.EtherCAT_Master_EPPxxxx.Beckhoff_EPP3xxx.Beckhoff_EPP3xxxEK1122.A_0006_EPP3184_0002_0018.AI_Standard_Channel_4.Status/Overrange <-> AI Standard Channel 4/Status/Overrange
//     PlcTask Inputs/GVL_iXlinker.EtherCAT_Master_EPPxxxx.Beckhoff_EPP3xxx.Beckhoff_EPP3xxxEK1122.A_0006_EPP3184_0002_0018.AI_Standard_Channel_1.Status/Limit_1 <-> AI Standard Channel 1/Status/Limit 1
//     PlcTask Inputs/GVL_iXlinker.EtherCAT_Master_EPPxxxx.Beckhoff_EPP3xxx.Beckhoff_EPP3xxxEK1122.A_0006_EPP3184_0002_0018.AI_Standard_Channel_1.Status/Limit_2 <-> AI Standard Channel 1/Status/Limit 2
//     PlcTask Inputs/GVL_iXlinker.EtherCAT_Master_EPPxxxx.Beckhoff_EPP3xxx.Beckhoff_EPP3xxxEK1122.A_0006_EPP3184_0002_0018.AI_Standard_Channel_2.Status/Limit_1 <-> AI Standard Channel 2/Status/Limit 1
//     PlcTask Inputs/GVL_iXlinker.EtherCAT_Master_EPPxxxx.Beckhoff_EPP3xxx.Beckhoff_EPP3xxxEK1122.A_0006_EPP3184_0002_0018.AI_Standard_Channel_2.Status/Limit_2 <-> AI Standard Channel 2/Status/Limit 2
//     PlcTask Inputs/GVL_iXlinker.EtherCAT_Master_EPPxxxx.Beckhoff_EPP3xxx.Beckhoff_EPP3xxxEK1122.A_0006_EPP3184_0002_0018.AI_Standard_Channel_3.Status/Limit_1 <-> AI Standard Channel 3/Status/Limit 1
//     PlcTask Inputs/GVL_iXlinker.EtherCAT_Master_EPPxxxx.Beckhoff_EPP3xxx.Beckhoff_EPP3xxxEK1122.A_0006_EPP3184_0002_0018.AI_Standard_Channel_3.Status/Limit_2 <-> AI Standard Channel 3/Status/Limit 2
//     PlcTask Inputs/GVL_iXlinker.EtherCAT_Master_EPPxxxx.Beckhoff_EPP3xxx.Beckhoff_EPP3xxxEK1122.A_0006_EPP3184_0002_0018.AI_Standard_Channel_4.Status/Limit_1 <-> AI Standard Channel 4/Status/Limit 1
//     PlcTask Inputs/GVL_iXlinker.EtherCAT_Master_EPPxxxx.Beckhoff_EPP3xxx.Beckhoff_EPP3xxxEK1122.A_0006_EPP3184_0002_0018.AI_Standard_Channel_4.Status/Limit_2 <-> AI Standard Channel 4/Status/Limit 2
//     PlcTask Inputs/GVL_iXlinker.EtherCAT_Master_EPPxxxx.Beckhoff_EPP3xxx.Beckhoff_EPP3xxxEK1122.A_0006_EPP3184_0002_0018.AI_Standard_Channel_1.Status/Error <-> AI Standard Channel 1/Status/Error
//     PlcTask Inputs/GVL_iXlinker.EtherCAT_Master_EPPxxxx.Beckhoff_EPP3xxx.Beckhoff_EPP3xxxEK1122.A_0006_EPP3184_0002_0018.AI_Standard_Channel_2.Status/Error <-> AI Standard Channel 2/Status/Error
//     PlcTask Inputs/GVL_iXlinker.EtherCAT_Master_EPPxxxx.Beckhoff_EPP3xxx.Beckhoff_EPP3xxxEK1122.A_0006_EPP3184_0002_0018.AI_Standard_Channel_3.Status/Error <-> AI Standard Channel 3/Status/Error
//     PlcTask Inputs/GVL_iXlinker.EtherCAT_Master_EPPxxxx.Beckhoff_EPP3xxx.Beckhoff_EPP3xxxEK1122.A_0006_EPP3184_0002_0018.AI_Standard_Channel_4.Status/Error <-> AI Standard Channel 4/Status/Error
//     PlcTask Inputs/GVL_iXlinker.EtherCAT_Master_EPPxxxx.Beckhoff_EPP3xxx.Beckhoff_EPP3xxxEK1122.A_0006_EPP3184_0002_0018.AI_Standard_Channel_1.Status/Sync_error <-> AI Standard Channel 1/Status/Sync error
//     PlcTask Inputs/GVL_iXlinker.EtherCAT_Master_EPPxxxx.Beckhoff_EPP3xxx.Beckhoff_EPP3xxxEK1122.A_0006_EPP3184_0002_0018.AI_Standard_Channel_2.Status/Sync_error <-> AI Standard Channel 2/Status/Sync error
//     PlcTask Inputs/GVL_iXlinker.EtherCAT_Master_EPPxxxx.Beckhoff_EPP3xxx.Beckhoff_EPP3xxxEK1122.A_0006_EPP3184_0002_0018.AI_Standard_Channel_3.Status/Sync_error <-> AI Standard Channel 3/Status/Sync error
//     PlcTask Inputs/GVL_iXlinker.EtherCAT_Master_EPPxxxx.Beckhoff_EPP3xxx.Beckhoff_EPP3xxxEK1122.A_0006_EPP3184_0002_0018.AI_Standard_Channel_4.Status/Sync_error <-> AI Standard Channel 4/Status/Sync error
//     PlcTask Inputs/GVL_iXlinker.EtherCAT_Master_EPPxxxx.Beckhoff_EPP3xxx.Beckhoff_EPP3xxxEK1122.A_0006_EPP3184_0002_0018.AI_Standard_Channel_1.Status/TxPDO_State <-> AI Standard Channel 1/Status/TxPDO State
//     PlcTask Inputs/GVL_iXlinker.EtherCAT_Master_EPPxxxx.Beckhoff_EPP3xxx.Beckhoff_EPP3xxxEK1122.A_0006_EPP3184_0002_0018.AI_Standard_Channel_2.Status/TxPDO_State <-> AI Standard Channel 2/Status/TxPDO State
//     PlcTask Inputs/GVL_iXlinker.EtherCAT_Master_EPPxxxx.Beckhoff_EPP3xxx.Beckhoff_EPP3xxxEK1122.A_0006_EPP3184_0002_0018.AI_Standard_Channel_3.Status/TxPDO_State <-> AI Standard Channel 3/Status/TxPDO State
//     PlcTask Inputs/GVL_iXlinker.EtherCAT_Master_EPPxxxx.Beckhoff_EPP3xxx.Beckhoff_EPP3xxxEK1122.A_0006_EPP3184_0002_0018.AI_Standard_Channel_4.Status/TxPDO_State <-> AI Standard Channel 4/Status/TxPDO State
//     PlcTask Inputs/GVL_iXlinker.EtherCAT_Master_EPPxxxx.Beckhoff_EPP3xxx.Beckhoff_EPP3xxxEK1122.A_0006_EPP3184_0002_0018.AI_Standard_Channel_1.Status/TxPDO_Toggle <-> AI Standard Channel 1/Status/TxPDO Toggle
//     PlcTask Inputs/GVL_iXlinker.EtherCAT_Master_EPPxxxx.Beckhoff_EPP3xxx.Beckhoff_EPP3xxxEK1122.A_0006_EPP3184_0002_0018.AI_Standard_Channel_2.Status/TxPDO_Toggle <-> AI Standard Channel 2/Status/TxPDO Toggle
//     PlcTask Inputs/GVL_iXlinker.EtherCAT_Master_EPPxxxx.Beckhoff_EPP3xxx.Beckhoff_EPP3xxxEK1122.A_0006_EPP3184_0002_0018.AI_Standard_Channel_3.Status/TxPDO_Toggle <-> AI Standard Channel 3/Status/TxPDO Toggle
//     PlcTask Inputs/GVL_iXlinker.EtherCAT_Master_EPPxxxx.Beckhoff_EPP3xxx.Beckhoff_EPP3xxxEK1122.A_0006_EPP3184_0002_0018.AI_Standard_Channel_4.Status/TxPDO_Toggle <-> AI Standard Channel 4/Status/TxPDO Toggle
//     PlcTask Inputs/GVL_iXlinker.EtherCAT_Master_EPPxxxx.Beckhoff_EPP3xxx.Beckhoff_EPP3xxxEK1122.A_0006_EPP3184_0002_0018.AI_Standard_Channel_1.Value <-> AI Standard Channel 1/Value
//     PlcTask Inputs/GVL_iXlinker.EtherCAT_Master_EPPxxxx.Beckhoff_EPP3xxx.Beckhoff_EPP3xxxEK1122.A_0006_EPP3184_0002_0018.AI_Standard_Channel_2.Value <-> AI Standard Channel 2/Value
//     PlcTask Inputs/GVL_iXlinker.EtherCAT_Master_EPPxxxx.Beckhoff_EPP3xxx.Beckhoff_EPP3xxxEK1122.A_0006_EPP3184_0002_0018.AI_Standard_Channel_3.Value <-> AI Standard Channel 3/Value
//     PlcTask Inputs/GVL_iXlinker.EtherCAT_Master_EPPxxxx.Beckhoff_EPP3xxx.Beckhoff_EPP3xxxEK1122.A_0006_EPP3184_0002_0018.AI_Standard_Channel_4.Value <-> AI Standard Channel 4/Value
//     PlcTask Inputs/GVL_iXlinker.EtherCAT_Master_EPPxxxx.Beckhoff_EPP3xxx.Beckhoff_EPP3xxxEK1122.A_0006_EPP3184_0002_0018.WcState.WcState <-> WcState/WcState
//     PlcTask Inputs/GVL_iXlinker.EtherCAT_Master_EPPxxxx.Beckhoff_EPP3xxx.Beckhoff_EPP3xxxEK1122.A_0006_EPP3184_0002_0018.WcState.InputToggle <-> WcState/InputToggle
//     PlcTask Inputs/GVL_iXlinker.EtherCAT_Master_EPPxxxx.Beckhoff_EPP3xxx.Beckhoff_EPP3xxxEK1122.A_0006_EPP3184_0002_0018.InfoData.AdsAddr <-> InfoData/AdsAddr
//     PlcTask Inputs/GVL_iXlinker.EtherCAT_Master_EPPxxxx.Beckhoff_EPP3xxx.Beckhoff_EPP3xxxEK1122.A_0006_EPP3184_0002_0018.InfoData.State <-> InfoData/State
//   PLC/PLC Instance <-> EtherCAT Master EPPxxxx/Beckhoff EPP3xxx/Beckhoff EPP3xxxEK1122/A_0007(EPP3184-0002-0019)
//     PlcTask Inputs/GVL_iXlinker.EtherCAT_Master_EPPxxxx.Beckhoff_EPP3xxx.Beckhoff_EPP3xxxEK1122.A_0007_EPP3184_0002_0019.AI_Standard_Channel_1.Status/Underrange <-> AI Standard Channel 1/Status/Underrange
//     PlcTask Inputs/GVL_iXlinker.EtherCAT_Master_EPPxxxx.Beckhoff_EPP3xxx.Beckhoff_EPP3xxxEK1122.A_0007_EPP3184_0002_0019.AI_Standard_Channel_2.Status/Underrange <-> AI Standard Channel 2/Status/Underrange
//     PlcTask Inputs/GVL_iXlinker.EtherCAT_Master_EPPxxxx.Beckhoff_EPP3xxx.Beckhoff_EPP3xxxEK1122.A_0007_EPP3184_0002_0019.AI_Standard_Channel_3.Status/Underrange <-> AI Standard Channel 3/Status/Underrange
//     PlcTask Inputs/GVL_iXlinker.EtherCAT_Master_EPPxxxx.Beckhoff_EPP3xxx.Beckhoff_EPP3xxxEK1122.A_0007_EPP3184_0002_0019.AI_Standard_Channel_4.Status/Underrange <-> AI Standard Channel 4/Status/Underrange
//     PlcTask Inputs/GVL_iXlinker.EtherCAT_Master_EPPxxxx.Beckhoff_EPP3xxx.Beckhoff_EPP3xxxEK1122.A_0007_EPP3184_0002_0019.AI_Standard_Channel_1.Status/Overrange <-> AI Standard Channel 1/Status/Overrange
//     PlcTask Inputs/GVL_iXlinker.EtherCAT_Master_EPPxxxx.Beckhoff_EPP3xxx.Beckhoff_EPP3xxxEK1122.A_0007_EPP3184_0002_0019.AI_Standard_Channel_2.Status/Overrange <-> AI Standard Channel 2/Status/Overrange
//     PlcTask Inputs/GVL_iXlinker.EtherCAT_Master_EPPxxxx.Beckhoff_EPP3xxx.Beckhoff_EPP3xxxEK1122.A_0007_EPP3184_0002_0019.AI_Standard_Channel_3.Status/Overrange <-> AI Standard Channel 3/Status/Overrange
//     PlcTask Inputs/GVL_iXlinker.EtherCAT_Master_EPPxxxx.Beckhoff_EPP3xxx.Beckhoff_EPP3xxxEK1122.A_0007_EPP3184_0002_0019.AI_Standard_Channel_4.Status/Overrange <-> AI Standard Channel 4/Status/Overrange
//     PlcTask Inputs/GVL_iXlinker.EtherCAT_Master_EPPxxxx.Beckhoff_EPP3xxx.Beckhoff_EPP3xxxEK1122.A_0007_EPP3184_0002_0019.AI_Standard_Channel_1.Status/Limit_1 <-> AI Standard Channel 1/Status/Limit 1
//     PlcTask Inputs/GVL_iXlinker.EtherCAT_Master_EPPxxxx.Beckhoff_EPP3xxx.Beckhoff_EPP3xxxEK1122.A_0007_EPP3184_0002_0019.AI_Standard_Channel_1.Status/Limit_2 <-> AI Standard Channel 1/Status/Limit 2
//     PlcTask Inputs/GVL_iXlinker.EtherCAT_Master_EPPxxxx.Beckhoff_EPP3xxx.Beckhoff_EPP3xxxEK1122.A_0007_EPP3184_0002_0019.AI_Standard_Channel_2.Status/Limit_1 <-> AI Standard Channel 2/Status/Limit 1
//     PlcTask Inputs/GVL_iXlinker.EtherCAT_Master_EPPxxxx.Beckhoff_EPP3xxx.Beckhoff_EPP3xxxEK1122.A_0007_EPP3184_0002_0019.AI_Standard_Channel_2.Status/Limit_2 <-> AI Standard Channel 2/Status/Limit 2
//     PlcTask Inputs/GVL_iXlinker.EtherCAT_Master_EPPxxxx.Beckhoff_EPP3xxx.Beckhoff_EPP3xxxEK1122.A_0007_EPP3184_0002_0019.AI_Standard_Channel_3.Status/Limit_1 <-> AI Standard Channel 3/Status/Limit 1
//     PlcTask Inputs/GVL_iXlinker.EtherCAT_Master_EPPxxxx.Beckhoff_EPP3xxx.Beckhoff_EPP3xxxEK1122.A_0007_EPP3184_0002_0019.AI_Standard_Channel_3.Status/Limit_2 <-> AI Standard Channel 3/Status/Limit 2
//     PlcTask Inputs/GVL_iXlinker.EtherCAT_Master_EPPxxxx.Beckhoff_EPP3xxx.Beckhoff_EPP3xxxEK1122.A_0007_EPP3184_0002_0019.AI_Standard_Channel_4.Status/Limit_1 <-> AI Standard Channel 4/Status/Limit 1
//     PlcTask Inputs/GVL_iXlinker.EtherCAT_Master_EPPxxxx.Beckhoff_EPP3xxx.Beckhoff_EPP3xxxEK1122.A_0007_EPP3184_0002_0019.AI_Standard_Channel_4.Status/Limit_2 <-> AI Standard Channel 4/Status/Limit 2
//     PlcTask Inputs/GVL_iXlinker.EtherCAT_Master_EPPxxxx.Beckhoff_EPP3xxx.Beckhoff_EPP3xxxEK1122.A_0007_EPP3184_0002_0019.AI_Standard_Channel_1.Status/Error <-> AI Standard Channel 1/Status/Error
//     PlcTask Inputs/GVL_iXlinker.EtherCAT_Master_EPPxxxx.Beckhoff_EPP3xxx.Beckhoff_EPP3xxxEK1122.A_0007_EPP3184_0002_0019.AI_Standard_Channel_2.Status/Error <-> AI Standard Channel 2/Status/Error
//     PlcTask Inputs/GVL_iXlinker.EtherCAT_Master_EPPxxxx.Beckhoff_EPP3xxx.Beckhoff_EPP3xxxEK1122.A_0007_EPP3184_0002_0019.AI_Standard_Channel_3.Status/Error <-> AI Standard Channel 3/Status/Error
//     PlcTask Inputs/GVL_iXlinker.EtherCAT_Master_EPPxxxx.Beckhoff_EPP3xxx.Beckhoff_EPP3xxxEK1122.A_0007_EPP3184_0002_0019.AI_Standard_Channel_4.Status/Error <-> AI Standard Channel 4/Status/Error
//     PlcTask Inputs/GVL_iXlinker.EtherCAT_Master_EPPxxxx.Beckhoff_EPP3xxx.Beckhoff_EPP3xxxEK1122.A_0007_EPP3184_0002_0019.AI_Standard_Channel_1.Status/Sync_error <-> AI Standard Channel 1/Status/Sync error
//     PlcTask Inputs/GVL_iXlinker.EtherCAT_Master_EPPxxxx.Beckhoff_EPP3xxx.Beckhoff_EPP3xxxEK1122.A_0007_EPP3184_0002_0019.AI_Standard_Channel_2.Status/Sync_error <-> AI Standard Channel 2/Status/Sync error
//     PlcTask Inputs/GVL_iXlinker.EtherCAT_Master_EPPxxxx.Beckhoff_EPP3xxx.Beckhoff_EPP3xxxEK1122.A_0007_EPP3184_0002_0019.AI_Standard_Channel_3.Status/Sync_error <-> AI Standard Channel 3/Status/Sync error
//     PlcTask Inputs/GVL_iXlinker.EtherCAT_Master_EPPxxxx.Beckhoff_EPP3xxx.Beckhoff_EPP3xxxEK1122.A_0007_EPP3184_0002_0019.AI_Standard_Channel_4.Status/Sync_error <-> AI Standard Channel 4/Status/Sync error
//     PlcTask Inputs/GVL_iXlinker.EtherCAT_Master_EPPxxxx.Beckhoff_EPP3xxx.Beckhoff_EPP3xxxEK1122.A_0007_EPP3184_0002_0019.AI_Standard_Channel_1.Status/TxPDO_State <-> AI Standard Channel 1/Status/TxPDO State
//     PlcTask Inputs/GVL_iXlinker.EtherCAT_Master_EPPxxxx.Beckhoff_EPP3xxx.Beckhoff_EPP3xxxEK1122.A_0007_EPP3184_0002_0019.AI_Standard_Channel_2.Status/TxPDO_State <-> AI Standard Channel 2/Status/TxPDO State
//     PlcTask Inputs/GVL_iXlinker.EtherCAT_Master_EPPxxxx.Beckhoff_EPP3xxx.Beckhoff_EPP3xxxEK1122.A_0007_EPP3184_0002_0019.AI_Standard_Channel_3.Status/TxPDO_State <-> AI Standard Channel 3/Status/TxPDO State
//     PlcTask Inputs/GVL_iXlinker.EtherCAT_Master_EPPxxxx.Beckhoff_EPP3xxx.Beckhoff_EPP3xxxEK1122.A_0007_EPP3184_0002_0019.AI_Standard_Channel_4.Status/TxPDO_State <-> AI Standard Channel 4/Status/TxPDO State
//     PlcTask Inputs/GVL_iXlinker.EtherCAT_Master_EPPxxxx.Beckhoff_EPP3xxx.Beckhoff_EPP3xxxEK1122.A_0007_EPP3184_0002_0019.AI_Standard_Channel_1.Status/TxPDO_Toggle <-> AI Standard Channel 1/Status/TxPDO Toggle
//     PlcTask Inputs/GVL_iXlinker.EtherCAT_Master_EPPxxxx.Beckhoff_EPP3xxx.Beckhoff_EPP3xxxEK1122.A_0007_EPP3184_0002_0019.AI_Standard_Channel_2.Status/TxPDO_Toggle <-> AI Standard Channel 2/Status/TxPDO Toggle
//     PlcTask Inputs/GVL_iXlinker.EtherCAT_Master_EPPxxxx.Beckhoff_EPP3xxx.Beckhoff_EPP3xxxEK1122.A_0007_EPP3184_0002_0019.AI_Standard_Channel_3.Status/TxPDO_Toggle <-> AI Standard Channel 3/Status/TxPDO Toggle
//     PlcTask Inputs/GVL_iXlinker.EtherCAT_Master_EPPxxxx.Beckhoff_EPP3xxx.Beckhoff_EPP3xxxEK1122.A_0007_EPP3184_0002_0019.AI_Standard_Channel_4.Status/TxPDO_Toggle <-> AI Standard Channel 4/Status/TxPDO Toggle
//     PlcTask Inputs/GVL_iXlinker.EtherCAT_Master_EPPxxxx.Beckhoff_EPP3xxx.Beckhoff_EPP3xxxEK1122.A_0007_EPP3184_0002_0019.AI_Standard_Channel_1.Value <-> AI Standard Channel 1/Value
//     PlcTask Inputs/GVL_iXlinker.EtherCAT_Master_EPPxxxx.Beckhoff_EPP3xxx.Beckhoff_EPP3xxxEK1122.A_0007_EPP3184_0002_0019.AI_Standard_Channel_2.Value <-> AI Standard Channel 2/Value
//     PlcTask Inputs/GVL_iXlinker.EtherCAT_Master_EPPxxxx.Beckhoff_EPP3xxx.Beckhoff_EPP3xxxEK1122.A_0007_EPP3184_0002_0019.AI_Standard_Channel_3.Value <-> AI Standard Channel 3/Value
//     PlcTask Inputs/GVL_iXlinker.EtherCAT_Master_EPPxxxx.Beckhoff_EPP3xxx.Beckhoff_EPP3xxxEK1122.A_0007_EPP3184_0002_0019.AI_Standard_Channel_4.Value <-> AI Standard Channel 4/Value
//     PlcTask Inputs/GVL_iXlinker.EtherCAT_Master_EPPxxxx.Beckhoff_EPP3xxx.Beckhoff_EPP3xxxEK1122.A_0007_EPP3184_0002_0019.WcState.WcState <-> WcState/WcState
//     PlcTask Inputs/GVL_iXlinker.EtherCAT_Master_EPPxxxx.Beckhoff_EPP3xxx.Beckhoff_EPP3xxxEK1122.A_0007_EPP3184_0002_0019.WcState.InputToggle <-> WcState/InputToggle
//     PlcTask Inputs/GVL_iXlinker.EtherCAT_Master_EPPxxxx.Beckhoff_EPP3xxx.Beckhoff_EPP3xxxEK1122.A_0007_EPP3184_0002_0019.InfoData.AdsAddr <-> InfoData/AdsAddr
//     PlcTask Inputs/GVL_iXlinker.EtherCAT_Master_EPPxxxx.Beckhoff_EPP3xxx.Beckhoff_EPP3xxxEK1122.A_0007_EPP3184_0002_0019.InfoData.State <-> InfoData/State
//   PLC/PLC Instance <-> EtherCAT Master EPPxxxx/Beckhoff EPP3xxx/Beckhoff EPP3xxxEK1122/A_0008(EPP3204-0002-0016)
//     PlcTask Inputs/GVL_iXlinker.EtherCAT_Master_EPPxxxx.Beckhoff_EPP3xxx.Beckhoff_EPP3xxxEK1122.A_0008_EPP3204_0002_0016.RTD_RTDInputs_Channel_1.Status/Underrange <-> RTD RTDInputs Channel 1/Status/Underrange
//     PlcTask Inputs/GVL_iXlinker.EtherCAT_Master_EPPxxxx.Beckhoff_EPP3xxx.Beckhoff_EPP3xxxEK1122.A_0008_EPP3204_0002_0016.RTD_RTDInputs_Channel_2.Status/Underrange <-> RTD RTDInputs Channel 2/Status/Underrange
//     PlcTask Inputs/GVL_iXlinker.EtherCAT_Master_EPPxxxx.Beckhoff_EPP3xxx.Beckhoff_EPP3xxxEK1122.A_0008_EPP3204_0002_0016.RTD_RTDInputs_Channel_3.Status/Underrange <-> RTD RTDInputs Channel 3/Status/Underrange
//     PlcTask Inputs/GVL_iXlinker.EtherCAT_Master_EPPxxxx.Beckhoff_EPP3xxx.Beckhoff_EPP3xxxEK1122.A_0008_EPP3204_0002_0016.RTD_RTDInputs_Channel_4.Status/Underrange <-> RTD RTDInputs Channel 4/Status/Underrange
//     PlcTask Inputs/GVL_iXlinker.EtherCAT_Master_EPPxxxx.Beckhoff_EPP3xxx.Beckhoff_EPP3xxxEK1122.A_0008_EPP3204_0002_0016.RTD_RTDInputs_Channel_1.Status/Overrange <-> RTD RTDInputs Channel 1/Status/Overrange
//     PlcTask Inputs/GVL_iXlinker.EtherCAT_Master_EPPxxxx.Beckhoff_EPP3xxx.Beckhoff_EPP3xxxEK1122.A_0008_EPP3204_0002_0016.RTD_RTDInputs_Channel_2.Status/Overrange <-> RTD RTDInputs Channel 2/Status/Overrange
//     PlcTask Inputs/GVL_iXlinker.EtherCAT_Master_EPPxxxx.Beckhoff_EPP3xxx.Beckhoff_EPP3xxxEK1122.A_0008_EPP3204_0002_0016.RTD_RTDInputs_Channel_3.Status/Overrange <-> RTD RTDInputs Channel 3/Status/Overrange
//     PlcTask Inputs/GVL_iXlinker.EtherCAT_Master_EPPxxxx.Beckhoff_EPP3xxx.Beckhoff_EPP3xxxEK1122.A_0008_EPP3204_0002_0016.RTD_RTDInputs_Channel_4.Status/Overrange <-> RTD RTDInputs Channel 4/Status/Overrange
//     PlcTask Inputs/GVL_iXlinker.EtherCAT_Master_EPPxxxx.Beckhoff_EPP3xxx.Beckhoff_EPP3xxxEK1122.A_0008_EPP3204_0002_0016.RTD_RTDInputs_Channel_1.Status/Limit_1 <-> RTD RTDInputs Channel 1/Status/Limit 1
//     PlcTask Inputs/GVL_iXlinker.EtherCAT_Master_EPPxxxx.Beckhoff_EPP3xxx.Beckhoff_EPP3xxxEK1122.A_0008_EPP3204_0002_0016.RTD_RTDInputs_Channel_1.Status/Limit_2 <-> RTD RTDInputs Channel 1/Status/Limit 2
//     PlcTask Inputs/GVL_iXlinker.EtherCAT_Master_EPPxxxx.Beckhoff_EPP3xxx.Beckhoff_EPP3xxxEK1122.A_0008_EPP3204_0002_0016.RTD_RTDInputs_Channel_2.Status/Limit_1 <-> RTD RTDInputs Channel 2/Status/Limit 1
//     PlcTask Inputs/GVL_iXlinker.EtherCAT_Master_EPPxxxx.Beckhoff_EPP3xxx.Beckhoff_EPP3xxxEK1122.A_0008_EPP3204_0002_0016.RTD_RTDInputs_Channel_2.Status/Limit_2 <-> RTD RTDInputs Channel 2/Status/Limit 2
//     PlcTask Inputs/GVL_iXlinker.EtherCAT_Master_EPPxxxx.Beckhoff_EPP3xxx.Beckhoff_EPP3xxxEK1122.A_0008_EPP3204_0002_0016.RTD_RTDInputs_Channel_3.Status/Limit_1 <-> RTD RTDInputs Channel 3/Status/Limit 1
//     PlcTask Inputs/GVL_iXlinker.EtherCAT_Master_EPPxxxx.Beckhoff_EPP3xxx.Beckhoff_EPP3xxxEK1122.A_0008_EPP3204_0002_0016.RTD_RTDInputs_Channel_3.Status/Limit_2 <-> RTD RTDInputs Channel 3/Status/Limit 2
//     PlcTask Inputs/GVL_iXlinker.EtherCAT_Master_EPPxxxx.Beckhoff_EPP3xxx.Beckhoff_EPP3xxxEK1122.A_0008_EPP3204_0002_0016.RTD_RTDInputs_Channel_4.Status/Limit_1 <-> RTD RTDInputs Channel 4/Status/Limit 1
//     PlcTask Inputs/GVL_iXlinker.EtherCAT_Master_EPPxxxx.Beckhoff_EPP3xxx.Beckhoff_EPP3xxxEK1122.A_0008_EPP3204_0002_0016.RTD_RTDInputs_Channel_4.Status/Limit_2 <-> RTD RTDInputs Channel 4/Status/Limit 2
//     PlcTask Inputs/GVL_iXlinker.EtherCAT_Master_EPPxxxx.Beckhoff_EPP3xxx.Beckhoff_EPP3xxxEK1122.A_0008_EPP3204_0002_0016.RTD_RTDInputs_Channel_1.Status/Error <-> RTD RTDInputs Channel 1/Status/Error
//     PlcTask Inputs/GVL_iXlinker.EtherCAT_Master_EPPxxxx.Beckhoff_EPP3xxx.Beckhoff_EPP3xxxEK1122.A_0008_EPP3204_0002_0016.RTD_RTDInputs_Channel_2.Status/Error <-> RTD RTDInputs Channel 2/Status/Error
//     PlcTask Inputs/GVL_iXlinker.EtherCAT_Master_EPPxxxx.Beckhoff_EPP3xxx.Beckhoff_EPP3xxxEK1122.A_0008_EPP3204_0002_0016.RTD_RTDInputs_Channel_3.Status/Error <-> RTD RTDInputs Channel 3/Status/Error
//     PlcTask Inputs/GVL_iXlinker.EtherCAT_Master_EPPxxxx.Beckhoff_EPP3xxx.Beckhoff_EPP3xxxEK1122.A_0008_EPP3204_0002_0016.RTD_RTDInputs_Channel_4.Status/Error <-> RTD RTDInputs Channel 4/Status/Error
//     PlcTask Inputs/GVL_iXlinker.EtherCAT_Master_EPPxxxx.Beckhoff_EPP3xxx.Beckhoff_EPP3xxxEK1122.A_0008_EPP3204_0002_0016.RTD_RTDInputs_Channel_1.Status/Sync_error <-> RTD RTDInputs Channel 1/Status/Sync error
//     PlcTask Inputs/GVL_iXlinker.EtherCAT_Master_EPPxxxx.Beckhoff_EPP3xxx.Beckhoff_EPP3xxxEK1122.A_0008_EPP3204_0002_0016.RTD_RTDInputs_Channel_2.Status/Sync_error <-> RTD RTDInputs Channel 2/Status/Sync error
//     PlcTask Inputs/GVL_iXlinker.EtherCAT_Master_EPPxxxx.Beckhoff_EPP3xxx.Beckhoff_EPP3xxxEK1122.A_0008_EPP3204_0002_0016.RTD_RTDInputs_Channel_3.Status/Sync_error <-> RTD RTDInputs Channel 3/Status/Sync error
//     PlcTask Inputs/GVL_iXlinker.EtherCAT_Master_EPPxxxx.Beckhoff_EPP3xxx.Beckhoff_EPP3xxxEK1122.A_0008_EPP3204_0002_0016.RTD_RTDInputs_Channel_4.Status/Sync_error <-> RTD RTDInputs Channel 4/Status/Sync error
//     PlcTask Inputs/GVL_iXlinker.EtherCAT_Master_EPPxxxx.Beckhoff_EPP3xxx.Beckhoff_EPP3xxxEK1122.A_0008_EPP3204_0002_0016.RTD_RTDInputs_Channel_1.Status/TxPDO_State <-> RTD RTDInputs Channel 1/Status/TxPDO State
//     PlcTask Inputs/GVL_iXlinker.EtherCAT_Master_EPPxxxx.Beckhoff_EPP3xxx.Beckhoff_EPP3xxxEK1122.A_0008_EPP3204_0002_0016.RTD_RTDInputs_Channel_2.Status/TxPDO_State <-> RTD RTDInputs Channel 2/Status/TxPDO State
//     PlcTask Inputs/GVL_iXlinker.EtherCAT_Master_EPPxxxx.Beckhoff_EPP3xxx.Beckhoff_EPP3xxxEK1122.A_0008_EPP3204_0002_0016.RTD_RTDInputs_Channel_3.Status/TxPDO_State <-> RTD RTDInputs Channel 3/Status/TxPDO State
//     PlcTask Inputs/GVL_iXlinker.EtherCAT_Master_EPPxxxx.Beckhoff_EPP3xxx.Beckhoff_EPP3xxxEK1122.A_0008_EPP3204_0002_0016.RTD_RTDInputs_Channel_4.Status/TxPDO_State <-> RTD RTDInputs Channel 4/Status/TxPDO State
//     PlcTask Inputs/GVL_iXlinker.EtherCAT_Master_EPPxxxx.Beckhoff_EPP3xxx.Beckhoff_EPP3xxxEK1122.A_0008_EPP3204_0002_0016.RTD_RTDInputs_Channel_1.Status/TxPDO_Toggle <-> RTD RTDInputs Channel 1/Status/TxPDO Toggle
//     PlcTask Inputs/GVL_iXlinker.EtherCAT_Master_EPPxxxx.Beckhoff_EPP3xxx.Beckhoff_EPP3xxxEK1122.A_0008_EPP3204_0002_0016.RTD_RTDInputs_Channel_2.Status/TxPDO_Toggle <-> RTD RTDInputs Channel 2/Status/TxPDO Toggle
//     PlcTask Inputs/GVL_iXlinker.EtherCAT_Master_EPPxxxx.Beckhoff_EPP3xxx.Beckhoff_EPP3xxxEK1122.A_0008_EPP3204_0002_0016.RTD_RTDInputs_Channel_3.Status/TxPDO_Toggle <-> RTD RTDInputs Channel 3/Status/TxPDO Toggle
//     PlcTask Inputs/GVL_iXlinker.EtherCAT_Master_EPPxxxx.Beckhoff_EPP3xxx.Beckhoff_EPP3xxxEK1122.A_0008_EPP3204_0002_0016.RTD_RTDInputs_Channel_4.Status/TxPDO_Toggle <-> RTD RTDInputs Channel 4/Status/TxPDO Toggle
//     PlcTask Inputs/GVL_iXlinker.EtherCAT_Master_EPPxxxx.Beckhoff_EPP3xxx.Beckhoff_EPP3xxxEK1122.A_0008_EPP3204_0002_0016.RTD_RTDInputs_Channel_1.Value <-> RTD RTDInputs Channel 1/Value
//     PlcTask Inputs/GVL_iXlinker.EtherCAT_Master_EPPxxxx.Beckhoff_EPP3xxx.Beckhoff_EPP3xxxEK1122.A_0008_EPP3204_0002_0016.RTD_RTDInputs_Channel_2.Value <-> RTD RTDInputs Channel 2/Value
//     PlcTask Inputs/GVL_iXlinker.EtherCAT_Master_EPPxxxx.Beckhoff_EPP3xxx.Beckhoff_EPP3xxxEK1122.A_0008_EPP3204_0002_0016.RTD_RTDInputs_Channel_3.Value <-> RTD RTDInputs Channel 3/Value
//     PlcTask Inputs/GVL_iXlinker.EtherCAT_Master_EPPxxxx.Beckhoff_EPP3xxx.Beckhoff_EPP3xxxEK1122.A_0008_EPP3204_0002_0016.RTD_RTDInputs_Channel_4.Value <-> RTD RTDInputs Channel 4/Value
//     PlcTask Inputs/GVL_iXlinker.EtherCAT_Master_EPPxxxx.Beckhoff_EPP3xxx.Beckhoff_EPP3xxxEK1122.A_0008_EPP3204_0002_0016.WcState.WcState <-> WcState/WcState
//     PlcTask Inputs/GVL_iXlinker.EtherCAT_Master_EPPxxxx.Beckhoff_EPP3xxx.Beckhoff_EPP3xxxEK1122.A_0008_EPP3204_0002_0016.WcState.InputToggle <-> WcState/InputToggle
//     PlcTask Inputs/GVL_iXlinker.EtherCAT_Master_EPPxxxx.Beckhoff_EPP3xxx.Beckhoff_EPP3xxxEK1122.A_0008_EPP3204_0002_0016.InfoData.AdsAddr <-> InfoData/AdsAddr
//     PlcTask Inputs/GVL_iXlinker.EtherCAT_Master_EPPxxxx.Beckhoff_EPP3xxx.Beckhoff_EPP3xxxEK1122.A_0008_EPP3204_0002_0016.InfoData.State <-> InfoData/State
//   PLC/PLC Instance <-> EtherCAT Master EPPxxxx/Beckhoff EPP3xxx/Beckhoff EPP3xxxEK1122/A_0009(EPP3204-0002-0017)
//     PlcTask Inputs/GVL_iXlinker.EtherCAT_Master_EPPxxxx.Beckhoff_EPP3xxx.Beckhoff_EPP3xxxEK1122.A_0009_EPP3204_0002_0017.RTD_RTDInputs_Channel_1.Status/Underrange <-> RTD RTDInputs Channel 1/Status/Underrange
//     PlcTask Inputs/GVL_iXlinker.EtherCAT_Master_EPPxxxx.Beckhoff_EPP3xxx.Beckhoff_EPP3xxxEK1122.A_0009_EPP3204_0002_0017.RTD_RTDInputs_Channel_2.Status/Underrange <-> RTD RTDInputs Channel 2/Status/Underrange
//     PlcTask Inputs/GVL_iXlinker.EtherCAT_Master_EPPxxxx.Beckhoff_EPP3xxx.Beckhoff_EPP3xxxEK1122.A_0009_EPP3204_0002_0017.RTD_RTDInputs_Channel_3.Status/Underrange <-> RTD RTDInputs Channel 3/Status/Underrange
//     PlcTask Inputs/GVL_iXlinker.EtherCAT_Master_EPPxxxx.Beckhoff_EPP3xxx.Beckhoff_EPP3xxxEK1122.A_0009_EPP3204_0002_0017.RTD_RTDInputs_Channel_4.Status/Underrange <-> RTD RTDInputs Channel 4/Status/Underrange
//     PlcTask Inputs/GVL_iXlinker.EtherCAT_Master_EPPxxxx.Beckhoff_EPP3xxx.Beckhoff_EPP3xxxEK1122.A_0009_EPP3204_0002_0017.RTD_RTDInputs_Channel_1.Status/Overrange <-> RTD RTDInputs Channel 1/Status/Overrange
//     PlcTask Inputs/GVL_iXlinker.EtherCAT_Master_EPPxxxx.Beckhoff_EPP3xxx.Beckhoff_EPP3xxxEK1122.A_0009_EPP3204_0002_0017.RTD_RTDInputs_Channel_2.Status/Overrange <-> RTD RTDInputs Channel 2/Status/Overrange
//     PlcTask Inputs/GVL_iXlinker.EtherCAT_Master_EPPxxxx.Beckhoff_EPP3xxx.Beckhoff_EPP3xxxEK1122.A_0009_EPP3204_0002_0017.RTD_RTDInputs_Channel_3.Status/Overrange <-> RTD RTDInputs Channel 3/Status/Overrange
//     PlcTask Inputs/GVL_iXlinker.EtherCAT_Master_EPPxxxx.Beckhoff_EPP3xxx.Beckhoff_EPP3xxxEK1122.A_0009_EPP3204_0002_0017.RTD_RTDInputs_Channel_4.Status/Overrange <-> RTD RTDInputs Channel 4/Status/Overrange
//     PlcTask Inputs/GVL_iXlinker.EtherCAT_Master_EPPxxxx.Beckhoff_EPP3xxx.Beckhoff_EPP3xxxEK1122.A_0009_EPP3204_0002_0017.RTD_RTDInputs_Channel_1.Status/Limit_1 <-> RTD RTDInputs Channel 1/Status/Limit 1
//     PlcTask Inputs/GVL_iXlinker.EtherCAT_Master_EPPxxxx.Beckhoff_EPP3xxx.Beckhoff_EPP3xxxEK1122.A_0009_EPP3204_0002_0017.RTD_RTDInputs_Channel_1.Status/Limit_2 <-> RTD RTDInputs Channel 1/Status/Limit 2
//     PlcTask Inputs/GVL_iXlinker.EtherCAT_Master_EPPxxxx.Beckhoff_EPP3xxx.Beckhoff_EPP3xxxEK1122.A_0009_EPP3204_0002_0017.RTD_RTDInputs_Channel_2.Status/Limit_1 <-> RTD RTDInputs Channel 2/Status/Limit 1
//     PlcTask Inputs/GVL_iXlinker.EtherCAT_Master_EPPxxxx.Beckhoff_EPP3xxx.Beckhoff_EPP3xxxEK1122.A_0009_EPP3204_0002_0017.RTD_RTDInputs_Channel_2.Status/Limit_2 <-> RTD RTDInputs Channel 2/Status/Limit 2
//     PlcTask Inputs/GVL_iXlinker.EtherCAT_Master_EPPxxxx.Beckhoff_EPP3xxx.Beckhoff_EPP3xxxEK1122.A_0009_EPP3204_0002_0017.RTD_RTDInputs_Channel_3.Status/Limit_1 <-> RTD RTDInputs Channel 3/Status/Limit 1
//     PlcTask Inputs/GVL_iXlinker.EtherCAT_Master_EPPxxxx.Beckhoff_EPP3xxx.Beckhoff_EPP3xxxEK1122.A_0009_EPP3204_0002_0017.RTD_RTDInputs_Channel_3.Status/Limit_2 <-> RTD RTDInputs Channel 3/Status/Limit 2
//     PlcTask Inputs/GVL_iXlinker.EtherCAT_Master_EPPxxxx.Beckhoff_EPP3xxx.Beckhoff_EPP3xxxEK1122.A_0009_EPP3204_0002_0017.RTD_RTDInputs_Channel_4.Status/Limit_1 <-> RTD RTDInputs Channel 4/Status/Limit 1
//     PlcTask Inputs/GVL_iXlinker.EtherCAT_Master_EPPxxxx.Beckhoff_EPP3xxx.Beckhoff_EPP3xxxEK1122.A_0009_EPP3204_0002_0017.RTD_RTDInputs_Channel_4.Status/Limit_2 <-> RTD RTDInputs Channel 4/Status/Limit 2
//     PlcTask Inputs/GVL_iXlinker.EtherCAT_Master_EPPxxxx.Beckhoff_EPP3xxx.Beckhoff_EPP3xxxEK1122.A_0009_EPP3204_0002_0017.RTD_RTDInputs_Channel_1.Status/Error <-> RTD RTDInputs Channel 1/Status/Error
//     PlcTask Inputs/GVL_iXlinker.EtherCAT_Master_EPPxxxx.Beckhoff_EPP3xxx.Beckhoff_EPP3xxxEK1122.A_0009_EPP3204_0002_0017.RTD_RTDInputs_Channel_2.Status/Error <-> RTD RTDInputs Channel 2/Status/Error
//     PlcTask Inputs/GVL_iXlinker.EtherCAT_Master_EPPxxxx.Beckhoff_EPP3xxx.Beckhoff_EPP3xxxEK1122.A_0009_EPP3204_0002_0017.RTD_RTDInputs_Channel_3.Status/Error <-> RTD RTDInputs Channel 3/Status/Error
//     PlcTask Inputs/GVL_iXlinker.EtherCAT_Master_EPPxxxx.Beckhoff_EPP3xxx.Beckhoff_EPP3xxxEK1122.A_0009_EPP3204_0002_0017.RTD_RTDInputs_Channel_4.Status/Error <-> RTD RTDInputs Channel 4/Status/Error
//     PlcTask Inputs/GVL_iXlinker.EtherCAT_Master_EPPxxxx.Beckhoff_EPP3xxx.Beckhoff_EPP3xxxEK1122.A_0009_EPP3204_0002_0017.RTD_RTDInputs_Channel_1.Status/TxPDO_State <-> RTD RTDInputs Channel 1/Status/TxPDO State
//     PlcTask Inputs/GVL_iXlinker.EtherCAT_Master_EPPxxxx.Beckhoff_EPP3xxx.Beckhoff_EPP3xxxEK1122.A_0009_EPP3204_0002_0017.RTD_RTDInputs_Channel_2.Status/TxPDO_State <-> RTD RTDInputs Channel 2/Status/TxPDO State
//     PlcTask Inputs/GVL_iXlinker.EtherCAT_Master_EPPxxxx.Beckhoff_EPP3xxx.Beckhoff_EPP3xxxEK1122.A_0009_EPP3204_0002_0017.RTD_RTDInputs_Channel_3.Status/TxPDO_State <-> RTD RTDInputs Channel 3/Status/TxPDO State
//     PlcTask Inputs/GVL_iXlinker.EtherCAT_Master_EPPxxxx.Beckhoff_EPP3xxx.Beckhoff_EPP3xxxEK1122.A_0009_EPP3204_0002_0017.RTD_RTDInputs_Channel_4.Status/TxPDO_State <-> RTD RTDInputs Channel 4/Status/TxPDO State
//     PlcTask Inputs/GVL_iXlinker.EtherCAT_Master_EPPxxxx.Beckhoff_EPP3xxx.Beckhoff_EPP3xxxEK1122.A_0009_EPP3204_0002_0017.RTD_RTDInputs_Channel_1.Status/TxPDO_Toggle <-> RTD RTDInputs Channel 1/Status/TxPDO Toggle
//     PlcTask Inputs/GVL_iXlinker.EtherCAT_Master_EPPxxxx.Beckhoff_EPP3xxx.Beckhoff_EPP3xxxEK1122.A_0009_EPP3204_0002_0017.RTD_RTDInputs_Channel_2.Status/TxPDO_Toggle <-> RTD RTDInputs Channel 2/Status/TxPDO Toggle
//     PlcTask Inputs/GVL_iXlinker.EtherCAT_Master_EPPxxxx.Beckhoff_EPP3xxx.Beckhoff_EPP3xxxEK1122.A_0009_EPP3204_0002_0017.RTD_RTDInputs_Channel_3.Status/TxPDO_Toggle <-> RTD RTDInputs Channel 3/Status/TxPDO Toggle
//     PlcTask Inputs/GVL_iXlinker.EtherCAT_Master_EPPxxxx.Beckhoff_EPP3xxx.Beckhoff_EPP3xxxEK1122.A_0009_EPP3204_0002_0017.RTD_RTDInputs_Channel_4.Status/TxPDO_Toggle <-> RTD RTDInputs Channel 4/Status/TxPDO Toggle
//     PlcTask Inputs/GVL_iXlinker.EtherCAT_Master_EPPxxxx.Beckhoff_EPP3xxx.Beckhoff_EPP3xxxEK1122.A_0009_EPP3204_0002_0017.RTD_RTDInputs_Channel_1.Value <-> RTD RTDInputs Channel 1/Value
//     PlcTask Inputs/GVL_iXlinker.EtherCAT_Master_EPPxxxx.Beckhoff_EPP3xxx.Beckhoff_EPP3xxxEK1122.A_0009_EPP3204_0002_0017.RTD_RTDInputs_Channel_2.Value <-> RTD RTDInputs Channel 2/Value
//     PlcTask Inputs/GVL_iXlinker.EtherCAT_Master_EPPxxxx.Beckhoff_EPP3xxx.Beckhoff_EPP3xxxEK1122.A_0009_EPP3204_0002_0017.RTD_RTDInputs_Channel_3.Value <-> RTD RTDInputs Channel 3/Value
//     PlcTask Inputs/GVL_iXlinker.EtherCAT_Master_EPPxxxx.Beckhoff_EPP3xxx.Beckhoff_EPP3xxxEK1122.A_0009_EPP3204_0002_0017.RTD_RTDInputs_Channel_4.Value <-> RTD RTDInputs Channel 4/Value
//     PlcTask Inputs/GVL_iXlinker.EtherCAT_Master_EPPxxxx.Beckhoff_EPP3xxx.Beckhoff_EPP3xxxEK1122.A_0009_EPP3204_0002_0017.WcState.WcState <-> WcState/WcState
//     PlcTask Inputs/GVL_iXlinker.EtherCAT_Master_EPPxxxx.Beckhoff_EPP3xxx.Beckhoff_EPP3xxxEK1122.A_0009_EPP3204_0002_0017.WcState.InputToggle <-> WcState/InputToggle
//     PlcTask Inputs/GVL_iXlinker.EtherCAT_Master_EPPxxxx.Beckhoff_EPP3xxx.Beckhoff_EPP3xxxEK1122.A_0009_EPP3204_0002_0017.InfoData.AdsAddr <-> InfoData/AdsAddr
//     PlcTask Inputs/GVL_iXlinker.EtherCAT_Master_EPPxxxx.Beckhoff_EPP3xxx.Beckhoff_EPP3xxxEK1122.A_0009_EPP3204_0002_0017.InfoData.State <-> InfoData/State
//   PLC/PLC Instance <-> EtherCAT Master EPPxxxx/Beckhoff EPP3xxx/Beckhoff EPP3xxxEK1122/A_0010(EPP3204-0002-0018)
//     PlcTask Inputs/GVL_iXlinker.EtherCAT_Master_EPPxxxx.Beckhoff_EPP3xxx.Beckhoff_EPP3xxxEK1122.A_0010_EPP3204_0002_0018.RTD_RTDInputs_Channel_1.Status/Underrange <-> RTD RTDInputs Channel 1/Status/Underrange
//     PlcTask Inputs/GVL_iXlinker.EtherCAT_Master_EPPxxxx.Beckhoff_EPP3xxx.Beckhoff_EPP3xxxEK1122.A_0010_EPP3204_0002_0018.RTD_RTDInputs_Channel_2.Status/Underrange <-> RTD RTDInputs Channel 2/Status/Underrange
//     PlcTask Inputs/GVL_iXlinker.EtherCAT_Master_EPPxxxx.Beckhoff_EPP3xxx.Beckhoff_EPP3xxxEK1122.A_0010_EPP3204_0002_0018.RTD_RTDInputs_Channel_3.Status/Underrange <-> RTD RTDInputs Channel 3/Status/Underrange
//     PlcTask Inputs/GVL_iXlinker.EtherCAT_Master_EPPxxxx.Beckhoff_EPP3xxx.Beckhoff_EPP3xxxEK1122.A_0010_EPP3204_0002_0018.RTD_RTDInputs_Channel_4.Status/Underrange <-> RTD RTDInputs Channel 4/Status/Underrange
//     PlcTask Inputs/GVL_iXlinker.EtherCAT_Master_EPPxxxx.Beckhoff_EPP3xxx.Beckhoff_EPP3xxxEK1122.A_0010_EPP3204_0002_0018.RTD_RTDInputs_Channel_1.Status/Overrange <-> RTD RTDInputs Channel 1/Status/Overrange
//     PlcTask Inputs/GVL_iXlinker.EtherCAT_Master_EPPxxxx.Beckhoff_EPP3xxx.Beckhoff_EPP3xxxEK1122.A_0010_EPP3204_0002_0018.RTD_RTDInputs_Channel_2.Status/Overrange <-> RTD RTDInputs Channel 2/Status/Overrange
//     PlcTask Inputs/GVL_iXlinker.EtherCAT_Master_EPPxxxx.Beckhoff_EPP3xxx.Beckhoff_EPP3xxxEK1122.A_0010_EPP3204_0002_0018.RTD_RTDInputs_Channel_3.Status/Overrange <-> RTD RTDInputs Channel 3/Status/Overrange
//     PlcTask Inputs/GVL_iXlinker.EtherCAT_Master_EPPxxxx.Beckhoff_EPP3xxx.Beckhoff_EPP3xxxEK1122.A_0010_EPP3204_0002_0018.RTD_RTDInputs_Channel_4.Status/Overrange <-> RTD RTDInputs Channel 4/Status/Overrange
//     PlcTask Inputs/GVL_iXlinker.EtherCAT_Master_EPPxxxx.Beckhoff_EPP3xxx.Beckhoff_EPP3xxxEK1122.A_0010_EPP3204_0002_0018.RTD_RTDInputs_Channel_1.Status/Limit_1 <-> RTD RTDInputs Channel 1/Status/Limit 1
//     PlcTask Inputs/GVL_iXlinker.EtherCAT_Master_EPPxxxx.Beckhoff_EPP3xxx.Beckhoff_EPP3xxxEK1122.A_0010_EPP3204_0002_0018.RTD_RTDInputs_Channel_1.Status/Limit_2 <-> RTD RTDInputs Channel 1/Status/Limit 2
//     PlcTask Inputs/GVL_iXlinker.EtherCAT_Master_EPPxxxx.Beckhoff_EPP3xxx.Beckhoff_EPP3xxxEK1122.A_0010_EPP3204_0002_0018.RTD_RTDInputs_Channel_2.Status/Limit_1 <-> RTD RTDInputs Channel 2/Status/Limit 1
//     PlcTask Inputs/GVL_iXlinker.EtherCAT_Master_EPPxxxx.Beckhoff_EPP3xxx.Beckhoff_EPP3xxxEK1122.A_0010_EPP3204_0002_0018.RTD_RTDInputs_Channel_2.Status/Limit_2 <-> RTD RTDInputs Channel 2/Status/Limit 2
//     PlcTask Inputs/GVL_iXlinker.EtherCAT_Master_EPPxxxx.Beckhoff_EPP3xxx.Beckhoff_EPP3xxxEK1122.A_0010_EPP3204_0002_0018.RTD_RTDInputs_Channel_3.Status/Limit_1 <-> RTD RTDInputs Channel 3/Status/Limit 1
//     PlcTask Inputs/GVL_iXlinker.EtherCAT_Master_EPPxxxx.Beckhoff_EPP3xxx.Beckhoff_EPP3xxxEK1122.A_0010_EPP3204_0002_0018.RTD_RTDInputs_Channel_3.Status/Limit_2 <-> RTD RTDInputs Channel 3/Status/Limit 2
//     PlcTask Inputs/GVL_iXlinker.EtherCAT_Master_EPPxxxx.Beckhoff_EPP3xxx.Beckhoff_EPP3xxxEK1122.A_0010_EPP3204_0002_0018.RTD_RTDInputs_Channel_4.Status/Limit_1 <-> RTD RTDInputs Channel 4/Status/Limit 1
//     PlcTask Inputs/GVL_iXlinker.EtherCAT_Master_EPPxxxx.Beckhoff_EPP3xxx.Beckhoff_EPP3xxxEK1122.A_0010_EPP3204_0002_0018.RTD_RTDInputs_Channel_4.Status/Limit_2 <-> RTD RTDInputs Channel 4/Status/Limit 2
//     PlcTask Inputs/GVL_iXlinker.EtherCAT_Master_EPPxxxx.Beckhoff_EPP3xxx.Beckhoff_EPP3xxxEK1122.A_0010_EPP3204_0002_0018.RTD_RTDInputs_Channel_1.Status/Error <-> RTD RTDInputs Channel 1/Status/Error
//     PlcTask Inputs/GVL_iXlinker.EtherCAT_Master_EPPxxxx.Beckhoff_EPP3xxx.Beckhoff_EPP3xxxEK1122.A_0010_EPP3204_0002_0018.RTD_RTDInputs_Channel_2.Status/Error <-> RTD RTDInputs Channel 2/Status/Error
//     PlcTask Inputs/GVL_iXlinker.EtherCAT_Master_EPPxxxx.Beckhoff_EPP3xxx.Beckhoff_EPP3xxxEK1122.A_0010_EPP3204_0002_0018.RTD_RTDInputs_Channel_3.Status/Error <-> RTD RTDInputs Channel 3/Status/Error
//     PlcTask Inputs/GVL_iXlinker.EtherCAT_Master_EPPxxxx.Beckhoff_EPP3xxx.Beckhoff_EPP3xxxEK1122.A_0010_EPP3204_0002_0018.RTD_RTDInputs_Channel_4.Status/Error <-> RTD RTDInputs Channel 4/Status/Error
//     PlcTask Inputs/GVL_iXlinker.EtherCAT_Master_EPPxxxx.Beckhoff_EPP3xxx.Beckhoff_EPP3xxxEK1122.A_0010_EPP3204_0002_0018.RTD_RTDInputs_Channel_1.Status/TxPDO_State <-> RTD RTDInputs Channel 1/Status/TxPDO State
//     PlcTask Inputs/GVL_iXlinker.EtherCAT_Master_EPPxxxx.Beckhoff_EPP3xxx.Beckhoff_EPP3xxxEK1122.A_0010_EPP3204_0002_0018.RTD_RTDInputs_Channel_2.Status/TxPDO_State <-> RTD RTDInputs Channel 2/Status/TxPDO State
//     PlcTask Inputs/GVL_iXlinker.EtherCAT_Master_EPPxxxx.Beckhoff_EPP3xxx.Beckhoff_EPP3xxxEK1122.A_0010_EPP3204_0002_0018.RTD_RTDInputs_Channel_3.Status/TxPDO_State <-> RTD RTDInputs Channel 3/Status/TxPDO State
//     PlcTask Inputs/GVL_iXlinker.EtherCAT_Master_EPPxxxx.Beckhoff_EPP3xxx.Beckhoff_EPP3xxxEK1122.A_0010_EPP3204_0002_0018.RTD_RTDInputs_Channel_4.Status/TxPDO_State <-> RTD RTDInputs Channel 4/Status/TxPDO State
//     PlcTask Inputs/GVL_iXlinker.EtherCAT_Master_EPPxxxx.Beckhoff_EPP3xxx.Beckhoff_EPP3xxxEK1122.A_0010_EPP3204_0002_0018.RTD_RTDInputs_Channel_1.Status/TxPDO_Toggle <-> RTD RTDInputs Channel 1/Status/TxPDO Toggle
//     PlcTask Inputs/GVL_iXlinker.EtherCAT_Master_EPPxxxx.Beckhoff_EPP3xxx.Beckhoff_EPP3xxxEK1122.A_0010_EPP3204_0002_0018.RTD_RTDInputs_Channel_2.Status/TxPDO_Toggle <-> RTD RTDInputs Channel 2/Status/TxPDO Toggle
//     PlcTask Inputs/GVL_iXlinker.EtherCAT_Master_EPPxxxx.Beckhoff_EPP3xxx.Beckhoff_EPP3xxxEK1122.A_0010_EPP3204_0002_0018.RTD_RTDInputs_Channel_3.Status/TxPDO_Toggle <-> RTD RTDInputs Channel 3/Status/TxPDO Toggle
//     PlcTask Inputs/GVL_iXlinker.EtherCAT_Master_EPPxxxx.Beckhoff_EPP3xxx.Beckhoff_EPP3xxxEK1122.A_0010_EPP3204_0002_0018.RTD_RTDInputs_Channel_4.Status/TxPDO_Toggle <-> RTD RTDInputs Channel 4/Status/TxPDO Toggle
//     PlcTask Inputs/GVL_iXlinker.EtherCAT_Master_EPPxxxx.Beckhoff_EPP3xxx.Beckhoff_EPP3xxxEK1122.A_0010_EPP3204_0002_0018.RTD_RTDInputs_Channel_1.Value <-> RTD RTDInputs Channel 1/Value
//     PlcTask Inputs/GVL_iXlinker.EtherCAT_Master_EPPxxxx.Beckhoff_EPP3xxx.Beckhoff_EPP3xxxEK1122.A_0010_EPP3204_0002_0018.RTD_RTDInputs_Channel_2.Value <-> RTD RTDInputs Channel 2/Value
//     PlcTask Inputs/GVL_iXlinker.EtherCAT_Master_EPPxxxx.Beckhoff_EPP3xxx.Beckhoff_EPP3xxxEK1122.A_0010_EPP3204_0002_0018.RTD_RTDInputs_Channel_3.Value <-> RTD RTDInputs Channel 3/Value
//     PlcTask Inputs/GVL_iXlinker.EtherCAT_Master_EPPxxxx.Beckhoff_EPP3xxx.Beckhoff_EPP3xxxEK1122.A_0010_EPP3204_0002_0018.RTD_RTDInputs_Channel_4.Value <-> RTD RTDInputs Channel 4/Value
//     PlcTask Inputs/GVL_iXlinker.EtherCAT_Master_EPPxxxx.Beckhoff_EPP3xxx.Beckhoff_EPP3xxxEK1122.A_0010_EPP3204_0002_0018.WcState.WcState <-> WcState/WcState
//     PlcTask Inputs/GVL_iXlinker.EtherCAT_Master_EPPxxxx.Beckhoff_EPP3xxx.Beckhoff_EPP3xxxEK1122.A_0010_EPP3204_0002_0018.WcState.InputToggle <-> WcState/InputToggle
//     PlcTask Inputs/GVL_iXlinker.EtherCAT_Master_EPPxxxx.Beckhoff_EPP3xxx.Beckhoff_EPP3xxxEK1122.A_0010_EPP3204_0002_0018.InfoData.AdsAddr <-> InfoData/AdsAddr
//     PlcTask Inputs/GVL_iXlinker.EtherCAT_Master_EPPxxxx.Beckhoff_EPP3xxx.Beckhoff_EPP3xxxEK1122.A_0010_EPP3204_0002_0018.InfoData.State <-> InfoData/State
//   PLC/PLC Instance <-> EtherCAT Master EPPxxxx/Beckhoff EPP3xxx/Beckhoff EPP3xxxEK1122/A_0011(EPP3204-0002-0019)
//     PlcTask Inputs/GVL_iXlinker.EtherCAT_Master_EPPxxxx.Beckhoff_EPP3xxx.Beckhoff_EPP3xxxEK1122.A_0011_EPP3204_0002_0019.RTD_RTDInputs_Channel_1.Status/Underrange <-> RTD RTDInputs Channel 1/Status/Underrange
//     PlcTask Inputs/GVL_iXlinker.EtherCAT_Master_EPPxxxx.Beckhoff_EPP3xxx.Beckhoff_EPP3xxxEK1122.A_0011_EPP3204_0002_0019.RTD_RTDInputs_Channel_2.Status/Underrange <-> RTD RTDInputs Channel 2/Status/Underrange
//     PlcTask Inputs/GVL_iXlinker.EtherCAT_Master_EPPxxxx.Beckhoff_EPP3xxx.Beckhoff_EPP3xxxEK1122.A_0011_EPP3204_0002_0019.RTD_RTDInputs_Channel_3.Status/Underrange <-> RTD RTDInputs Channel 3/Status/Underrange
//     PlcTask Inputs/GVL_iXlinker.EtherCAT_Master_EPPxxxx.Beckhoff_EPP3xxx.Beckhoff_EPP3xxxEK1122.A_0011_EPP3204_0002_0019.RTD_RTDInputs_Channel_4.Status/Underrange <-> RTD RTDInputs Channel 4/Status/Underrange
//     PlcTask Inputs/GVL_iXlinker.EtherCAT_Master_EPPxxxx.Beckhoff_EPP3xxx.Beckhoff_EPP3xxxEK1122.A_0011_EPP3204_0002_0019.RTD_RTDInputs_Channel_1.Status/Overrange <-> RTD RTDInputs Channel 1/Status/Overrange
//     PlcTask Inputs/GVL_iXlinker.EtherCAT_Master_EPPxxxx.Beckhoff_EPP3xxx.Beckhoff_EPP3xxxEK1122.A_0011_EPP3204_0002_0019.RTD_RTDInputs_Channel_2.Status/Overrange <-> RTD RTDInputs Channel 2/Status/Overrange
//     PlcTask Inputs/GVL_iXlinker.EtherCAT_Master_EPPxxxx.Beckhoff_EPP3xxx.Beckhoff_EPP3xxxEK1122.A_0011_EPP3204_0002_0019.RTD_RTDInputs_Channel_3.Status/Overrange <-> RTD RTDInputs Channel 3/Status/Overrange
//     PlcTask Inputs/GVL_iXlinker.EtherCAT_Master_EPPxxxx.Beckhoff_EPP3xxx.Beckhoff_EPP3xxxEK1122.A_0011_EPP3204_0002_0019.RTD_RTDInputs_Channel_4.Status/Overrange <-> RTD RTDInputs Channel 4/Status/Overrange
//     PlcTask Inputs/GVL_iXlinker.EtherCAT_Master_EPPxxxx.Beckhoff_EPP3xxx.Beckhoff_EPP3xxxEK1122.A_0011_EPP3204_0002_0019.RTD_RTDInputs_Channel_1.Status/Limit_1 <-> RTD RTDInputs Channel 1/Status/Limit 1
//     PlcTask Inputs/GVL_iXlinker.EtherCAT_Master_EPPxxxx.Beckhoff_EPP3xxx.Beckhoff_EPP3xxxEK1122.A_0011_EPP3204_0002_0019.RTD_RTDInputs_Channel_1.Status/Limit_2 <-> RTD RTDInputs Channel 1/Status/Limit 2
//     PlcTask Inputs/GVL_iXlinker.EtherCAT_Master_EPPxxxx.Beckhoff_EPP3xxx.Beckhoff_EPP3xxxEK1122.A_0011_EPP3204_0002_0019.RTD_RTDInputs_Channel_2.Status/Limit_1 <-> RTD RTDInputs Channel 2/Status/Limit 1
//     PlcTask Inputs/GVL_iXlinker.EtherCAT_Master_EPPxxxx.Beckhoff_EPP3xxx.Beckhoff_EPP3xxxEK1122.A_0011_EPP3204_0002_0019.RTD_RTDInputs_Channel_2.Status/Limit_2 <-> RTD RTDInputs Channel 2/Status/Limit 2
//     PlcTask Inputs/GVL_iXlinker.EtherCAT_Master_EPPxxxx.Beckhoff_EPP3xxx.Beckhoff_EPP3xxxEK1122.A_0011_EPP3204_0002_0019.RTD_RTDInputs_Channel_3.Status/Limit_1 <-> RTD RTDInputs Channel 3/Status/Limit 1
//     PlcTask Inputs/GVL_iXlinker.EtherCAT_Master_EPPxxxx.Beckhoff_EPP3xxx.Beckhoff_EPP3xxxEK1122.A_0011_EPP3204_0002_0019.RTD_RTDInputs_Channel_3.Status/Limit_2 <-> RTD RTDInputs Channel 3/Status/Limit 2
//     PlcTask Inputs/GVL_iXlinker.EtherCAT_Master_EPPxxxx.Beckhoff_EPP3xxx.Beckhoff_EPP3xxxEK1122.A_0011_EPP3204_0002_0019.RTD_RTDInputs_Channel_4.Status/Limit_1 <-> RTD RTDInputs Channel 4/Status/Limit 1
//     PlcTask Inputs/GVL_iXlinker.EtherCAT_Master_EPPxxxx.Beckhoff_EPP3xxx.Beckhoff_EPP3xxxEK1122.A_0011_EPP3204_0002_0019.RTD_RTDInputs_Channel_4.Status/Limit_2 <-> RTD RTDInputs Channel 4/Status/Limit 2
//     PlcTask Inputs/GVL_iXlinker.EtherCAT_Master_EPPxxxx.Beckhoff_EPP3xxx.Beckhoff_EPP3xxxEK1122.A_0011_EPP3204_0002_0019.RTD_RTDInputs_Channel_1.Status/Error <-> RTD RTDInputs Channel 1/Status/Error
//     PlcTask Inputs/GVL_iXlinker.EtherCAT_Master_EPPxxxx.Beckhoff_EPP3xxx.Beckhoff_EPP3xxxEK1122.A_0011_EPP3204_0002_0019.RTD_RTDInputs_Channel_2.Status/Error <-> RTD RTDInputs Channel 2/Status/Error
//     PlcTask Inputs/GVL_iXlinker.EtherCAT_Master_EPPxxxx.Beckhoff_EPP3xxx.Beckhoff_EPP3xxxEK1122.A_0011_EPP3204_0002_0019.RTD_RTDInputs_Channel_3.Status/Error <-> RTD RTDInputs Channel 3/Status/Error
//     PlcTask Inputs/GVL_iXlinker.EtherCAT_Master_EPPxxxx.Beckhoff_EPP3xxx.Beckhoff_EPP3xxxEK1122.A_0011_EPP3204_0002_0019.RTD_RTDInputs_Channel_4.Status/Error <-> RTD RTDInputs Channel 4/Status/Error
//     PlcTask Inputs/GVL_iXlinker.EtherCAT_Master_EPPxxxx.Beckhoff_EPP3xxx.Beckhoff_EPP3xxxEK1122.A_0011_EPP3204_0002_0019.RTD_RTDInputs_Channel_1.Status/TxPDO_State <-> RTD RTDInputs Channel 1/Status/TxPDO State
//     PlcTask Inputs/GVL_iXlinker.EtherCAT_Master_EPPxxxx.Beckhoff_EPP3xxx.Beckhoff_EPP3xxxEK1122.A_0011_EPP3204_0002_0019.RTD_RTDInputs_Channel_2.Status/TxPDO_State <-> RTD RTDInputs Channel 2/Status/TxPDO State
//     PlcTask Inputs/GVL_iXlinker.EtherCAT_Master_EPPxxxx.Beckhoff_EPP3xxx.Beckhoff_EPP3xxxEK1122.A_0011_EPP3204_0002_0019.RTD_RTDInputs_Channel_3.Status/TxPDO_State <-> RTD RTDInputs Channel 3/Status/TxPDO State
//     PlcTask Inputs/GVL_iXlinker.EtherCAT_Master_EPPxxxx.Beckhoff_EPP3xxx.Beckhoff_EPP3xxxEK1122.A_0011_EPP3204_0002_0019.RTD_RTDInputs_Channel_4.Status/TxPDO_State <-> RTD RTDInputs Channel 4/Status/TxPDO State
//     PlcTask Inputs/GVL_iXlinker.EtherCAT_Master_EPPxxxx.Beckhoff_EPP3xxx.Beckhoff_EPP3xxxEK1122.A_0011_EPP3204_0002_0019.RTD_RTDInputs_Channel_1.Status/TxPDO_Toggle <-> RTD RTDInputs Channel 1/Status/TxPDO Toggle
//     PlcTask Inputs/GVL_iXlinker.EtherCAT_Master_EPPxxxx.Beckhoff_EPP3xxx.Beckhoff_EPP3xxxEK1122.A_0011_EPP3204_0002_0019.RTD_RTDInputs_Channel_2.Status/TxPDO_Toggle <-> RTD RTDInputs Channel 2/Status/TxPDO Toggle
//     PlcTask Inputs/GVL_iXlinker.EtherCAT_Master_EPPxxxx.Beckhoff_EPP3xxx.Beckhoff_EPP3xxxEK1122.A_0011_EPP3204_0002_0019.RTD_RTDInputs_Channel_3.Status/TxPDO_Toggle <-> RTD RTDInputs Channel 3/Status/TxPDO Toggle
//     PlcTask Inputs/GVL_iXlinker.EtherCAT_Master_EPPxxxx.Beckhoff_EPP3xxx.Beckhoff_EPP3xxxEK1122.A_0011_EPP3204_0002_0019.RTD_RTDInputs_Channel_4.Status/TxPDO_Toggle <-> RTD RTDInputs Channel 4/Status/TxPDO Toggle
//     PlcTask Inputs/GVL_iXlinker.EtherCAT_Master_EPPxxxx.Beckhoff_EPP3xxx.Beckhoff_EPP3xxxEK1122.A_0011_EPP3204_0002_0019.RTD_RTDInputs_Channel_1.Value <-> RTD RTDInputs Channel 1/Value
//     PlcTask Inputs/GVL_iXlinker.EtherCAT_Master_EPPxxxx.Beckhoff_EPP3xxx.Beckhoff_EPP3xxxEK1122.A_0011_EPP3204_0002_0019.RTD_RTDInputs_Channel_2.Value <-> RTD RTDInputs Channel 2/Value
//     PlcTask Inputs/GVL_iXlinker.EtherCAT_Master_EPPxxxx.Beckhoff_EPP3xxx.Beckhoff_EPP3xxxEK1122.A_0011_EPP3204_0002_0019.RTD_RTDInputs_Channel_3.Value <-> RTD RTDInputs Channel 3/Value
//     PlcTask Inputs/GVL_iXlinker.EtherCAT_Master_EPPxxxx.Beckhoff_EPP3xxx.Beckhoff_EPP3xxxEK1122.A_0011_EPP3204_0002_0019.RTD_RTDInputs_Channel_4.Value <-> RTD RTDInputs Channel 4/Value
//     PlcTask Inputs/GVL_iXlinker.EtherCAT_Master_EPPxxxx.Beckhoff_EPP3xxx.Beckhoff_EPP3xxxEK1122.A_0011_EPP3204_0002_0019.WcState.WcState <-> WcState/WcState
//     PlcTask Inputs/GVL_iXlinker.EtherCAT_Master_EPPxxxx.Beckhoff_EPP3xxx.Beckhoff_EPP3xxxEK1122.A_0011_EPP3204_0002_0019.WcState.InputToggle <-> WcState/InputToggle
//     PlcTask Inputs/GVL_iXlinker.EtherCAT_Master_EPPxxxx.Beckhoff_EPP3xxx.Beckhoff_EPP3xxxEK1122.A_0011_EPP3204_0002_0019.InfoData.AdsAddr <-> InfoData/AdsAddr
//     PlcTask Inputs/GVL_iXlinker.EtherCAT_Master_EPPxxxx.Beckhoff_EPP3xxx.Beckhoff_EPP3xxxEK1122.A_0011_EPP3204_0002_0019.InfoData.State <-> InfoData/State
//   PLC/PLC Instance <-> EtherCAT Master EPPxxxx/Beckhoff EPP3xxx/Beckhoff EPP3xxxEK1122/A_0012(EPP3314-0002-0016)
//     PlcTask Inputs/GVL_iXlinker.EtherCAT_Master_EPPxxxx.Beckhoff_EPP3xxx.Beckhoff_EPP3xxxEK1122.A_0012_EPP3314_0002_0016.TC_Inputs_Channel_1.Status/Underrange <-> TC Inputs Channel 1/Status/Underrange
//     PlcTask Inputs/GVL_iXlinker.EtherCAT_Master_EPPxxxx.Beckhoff_EPP3xxx.Beckhoff_EPP3xxxEK1122.A_0012_EPP3314_0002_0016.TC_Inputs_Channel_2.Status/Underrange <-> TC Inputs Channel 2/Status/Underrange
//     PlcTask Inputs/GVL_iXlinker.EtherCAT_Master_EPPxxxx.Beckhoff_EPP3xxx.Beckhoff_EPP3xxxEK1122.A_0012_EPP3314_0002_0016.TC_Inputs_Channel_3.Status/Underrange <-> TC Inputs Channel 3/Status/Underrange
//     PlcTask Inputs/GVL_iXlinker.EtherCAT_Master_EPPxxxx.Beckhoff_EPP3xxx.Beckhoff_EPP3xxxEK1122.A_0012_EPP3314_0002_0016.TC_Inputs_Channel_4.Status/Underrange <-> TC Inputs Channel 4/Status/Underrange
//     PlcTask Inputs/GVL_iXlinker.EtherCAT_Master_EPPxxxx.Beckhoff_EPP3xxx.Beckhoff_EPP3xxxEK1122.A_0012_EPP3314_0002_0016.TC_Inputs_Channel_1.Status/Overrange <-> TC Inputs Channel 1/Status/Overrange
//     PlcTask Inputs/GVL_iXlinker.EtherCAT_Master_EPPxxxx.Beckhoff_EPP3xxx.Beckhoff_EPP3xxxEK1122.A_0012_EPP3314_0002_0016.TC_Inputs_Channel_2.Status/Overrange <-> TC Inputs Channel 2/Status/Overrange
//     PlcTask Inputs/GVL_iXlinker.EtherCAT_Master_EPPxxxx.Beckhoff_EPP3xxx.Beckhoff_EPP3xxxEK1122.A_0012_EPP3314_0002_0016.TC_Inputs_Channel_3.Status/Overrange <-> TC Inputs Channel 3/Status/Overrange
//     PlcTask Inputs/GVL_iXlinker.EtherCAT_Master_EPPxxxx.Beckhoff_EPP3xxx.Beckhoff_EPP3xxxEK1122.A_0012_EPP3314_0002_0016.TC_Inputs_Channel_4.Status/Overrange <-> TC Inputs Channel 4/Status/Overrange
//     PlcTask Inputs/GVL_iXlinker.EtherCAT_Master_EPPxxxx.Beckhoff_EPP3xxx.Beckhoff_EPP3xxxEK1122.A_0012_EPP3314_0002_0016.TC_Inputs_Channel_1.Status/Limit_1 <-> TC Inputs Channel 1/Status/Limit 1
